LIN {X 0,Y 297.414,Z 212.275,A -85,B 0,C 180,E1 -16492.846,E2 -16492.846} C_VEL
LIN {X 0,Y 297.108,Z 216.721,A -85,B 0,C 180,E1 -16496.707,E2 -16496.707} C_VEL
LIN {X 0,Y 297.039,Z 218.831,A -85,B 0,C 180,E1 -16498.514,E2 -16498.514} C_VEL
LIN {X 0,Y 298.985,Z 230.293,A -85,B 0,C 180,E1 -16499.329,E2 -16499.329} C_VEL
LIN {X 0,Y 300.063,Z 238.045,A -85,B 0,C 180,E1 -16500.022,E2 -16500.022} C_VEL
LIN {X 0,Y 300.785,Z 244.745,A -85,B 0,C 180,E1 -16500.738,E2 -16500.738} C_VEL
LIN {X 0,Y 300.112,Z 253.295,A -85,B 0,C 180,E1 -16501.796,E2 -16501.796} C_VEL
LIN {X 0,Y 299.342,Z 261.65,A -85,B 0,C 180,E1 -16503.084,E2 -16503.084} C_VEL
LIN {X 0,Y 298.596,Z 269.147,A -85,B 0,C 180,E1 -16504.537,E2 -16504.537} C_VEL
LIN {X 0,Y 298.008,Z 275.588,A -85,B 0,C 180,E1 -16506.127,E2 -16506.127} C_VEL
LIN {X 0,Y 297.4,Z 281.322,A -85,B 0,C 180,E1 -16507.91,E2 -16507.91} C_VEL
LIN {X 0,Y 296.932,Z 285.817,A -85,B 0,C 180,E1 -16509.721,E2 -16509.721} C_VEL
LIN {X 0,Y 296.668,Z 289.117,A -85,B 0,C 180,E1 -16511.553,E2 -16511.553} C_VEL
LIN {X 0,Y 296.474,Z 291.311,A -85,B 0,C 180,E1 -16513.429,E2 -16513.429} C_VEL
LIN {X 0,Y 296.443,Z 292.469,A -85,B 0,C 180,E1 -16515.335,E2 -16515.335} C_VEL
LIN {X 0,Y 296.588,Z 292.583,A -85,B 0,C 180,E1 -16517.272,E2 -16517.272} C_VEL
LIN {X 0,Y 296.965,Z 291.615,A -85,B 0,C 180,E1 -16519.228,E2 -16519.228} C_VEL
LIN {X 0,Y 297.538,Z 289.488,A -85,B 0,C 180,E1 -16521.212,E2 -16521.212} C_VEL
LIN {X 0,Y 298.269,Z 285.912,A -85,B 0,C 180,E1 -16523.238,E2 -16523.238} C_VEL
LIN {X 0,Y 299.253,Z 280.84,A -85,B 0,C 180,E1 -16525.283,E2 -16525.283} C_VEL
LIN {X 0,Y 300.568,Z 273.927,A -85,B 0,C 180,E1 -16527.327,E2 -16527.327} C_VEL
LIN {X 0,Y 301.642,Z 267.542,A -85,B 0,C 180,E1 -16528.776,E2 -16528.776} C_VEL
LIN {X 0,Y 302.836,Z 260.472,A -85,B 0,C 180,E1 -16530.071,E2 -16530.071} C_VEL
LIN {X 0,Y 304.08,Z 251.263,A -85,B 0,C 180,E1 -16531.434,E2 -16531.434} C_VEL
LIN {X 0,Y 303.978,Z 248.011,A -85,B 0,C 180,E1 -16531.86,E2 -16531.86} C_VEL
LIN {X 0,Y 302.759,Z 239.813,A -85,B 0,C 180,E1 -16532.901,E2 -16532.901} C_VEL
LIN {X 0,Y 301.269,Z 232.79,A -85,B 0,C 180,E1 -16533.691,E2 -16533.691} C_VEL
LIN {X 0,Y 298.786,Z 224.127,A -85,B 0,C 180,E1 -16534.557,E2 -16534.557} C_VEL
LIN {X 0,Y 297.767,Z 220.447,A -85,B 0,C 180,E1 -16534.908,E2 -16534.908} C_VEL
LIN {X 0,Y 298.166,Z 216.073,A -85,B 0,C 180,E1 -16539.296,E2 -16539.296} C_VEL
LIN {X 0,Y 298.502,Z 213.292,A -85,B 0,C 180,E1 -16542.179,E2 -16542.179} C_VEL
LIN {X 0,Y 298.837,Z 210.683,A -85,B 0,C 180,E1 -16545.009,E2 -16545.009} C_VEL
LIN {X 0,Y 298.987,Z 208.224,A -85,B 0,C 180,E1 -16547.788,E2 -16547.788} C_VEL
LIN {X 0,Y 298.888,Z 204.918,A -85,B 0,C 180,E1 -16551.891,E2 -16551.891} C_VEL
LIN {X 0,Y 298.802,Z 204.086,A -85,B 0,C 180,E1 -16553.247,E2 -16553.247} C_VEL
LIN {X 0,Y 298.84,Z 204.074,A -85,B 0,C 180,E1 -16557.531,E2 -16557.531} C_VEL
LIN {X 0,Y 298.211,Z 204.153,A -85,B 0,C 180,E1 -16558.658,E2 -16558.658} C_VEL
LIN {X 0,Y 295.396,Z 204.503,A -85,B 0,C 180,E1 -16560.493,E2 -16560.493} C_VEL
LIN {X 0,Y 292.054,Z 204.917,A -85,B 0,C 180,E1 -16562.745,E2 -16562.745} C_VEL
LIN {X 0,Y 291.638,Z 204.968,A -85,B 0,C 180,E1 -16563.524,E2 -16563.524} C_VEL
LIN {X 0,Y 291.725,Z 204.961,A -85,B 0,C 180,E1 -16566.92,E2 -16566.92} C_VEL
LIN {X 0,Y 291.569,Z 204.98,A -85,B 0,C 180,E1 -16569.715,E2 -16569.715} C_VEL
LIN {X 0,Y 291.524,Z 204.986,A -85,B 0,C 180,E1 -16573.951,E2 -16573.951} C_VEL
LIN {X 0,Y 291.489,Z 204.99,A -85,B 0,C 180,E1 -16576.819,E2 -16576.819} C_VEL
LIN {X 0,Y 291.453,Z 204.994,A -85,B 0,C 180,E1 -16579.876,E2 -16579.876} C_VEL
LIN {X 0,Y 291.403,Z 205.001,A -85,B 0,C 180,E1 -16584.206,E2 -16584.206} C_VEL
LIN {X 0,Y 291.425,Z 204.997,A -85,B 0,C 180,E1 -16587.272,E2 -16587.272} C_VEL
LIN {X 0,Y 291.34,Z 205.007,A -85,B 0,C 180,E1 -16590.438,E2 -16590.438} C_VEL
LIN {X 0,Y 291.347,Z 205.006,A -85,B 0,C 180,E1 -16593.699,E2 -16593.699} C_VEL
LIN {X 0,Y 291.383,Z 205.003,A -85,B 0,C 180,E1 -16597.256,E2 -16597.256} C_VEL
LIN {X 0,Y 291.336,Z 205.011,A -85,B 0,C 180,E1 -16600.643,E2 -16600.643} C_VEL
LIN {X 0,Y 291.356,Z 205.078,A -85,B 0,C 180,E1 -16602.79,E2 -16602.79} C_VEL
LIN {X 0,Y 291.895,Z 208.233,A -85,B 0,C 180,E1 -16606.247,E2 -16606.247} C_VEL
LIN {X 0,Y 292.713,Z 212.344,A -85,B 0,C 180,E1 -16610.204,E2 -16610.204} C_VEL
LIN {X 0,Y 293.351,Z 215.803,A -85,B 0,C 180,E1 -16613.206,E2 -16613.206} C_VEL
LIN {X 0,Y 294.12,Z 220.258,A -85,B 0,C 180,E1 -16616.755,E2 -16616.755} C_VEL
LIN {X 0,Y 294.047,Z 222.378,A -85,B 0,C 180,E1 -16618.277,E2 -16618.277} C_VEL
LIN {X 0,Y 293.07,Z 226.935,A -85,B 0,C 180,E1 -16621.34,E2 -16621.34} C_VEL
LIN {X 0,Y 291.758,Z 233.962,A -85,B 0,C 180,E1 -16625.827,E2 -16625.827} C_VEL
LIN {X 0,Y 291.109,Z 238.512,A -85,B 0,C 180,E1 -16628.63,E2 -16628.63} C_VEL
LIN {X 0,Y 293.61,Z 250.168,A -85,B 0,C 180,E1 -16629.573,E2 -16629.573} C_VEL
LIN {X 0,Y 295.041,Z 259.692,A -85,B 0,C 180,E1 -16630.52,E2 -16630.52} C_VEL
LIN {X 0,Y 295.682,Z 269.392,A -85,B 0,C 180,E1 -16631.644,E2 -16631.644} C_VEL
LIN {X 0,Y 295.708,Z 276.379,A -85,B 0,C 180,E1 -16632.581,E2 -16632.581} C_VEL
LIN {X 0,Y 295.117,Z 282.939,A -85,B 0,C 180,E1 -16633.573,E2 -16633.573} C_VEL
LIN {X 0,Y 293.912,Z 289.657,A -85,B 0,C 180,E1 -16634.75,E2 -16634.75} C_VEL
LIN {X 0,Y 292.758,Z 296.048,A -85,B 0,C 180,E1 -16636.11,E2 -16636.11} C_VEL
LIN {X 0,Y 291.865,Z 301.377,A -85,B 0,C 180,E1 -16637.484,E2 -16637.484} C_VEL
LIN {X 0,Y 291.099,Z 305.839,A -85,B 0,C 180,E1 -16638.864,E2 -16638.864} C_VEL
LIN {X 0,Y 290.259,Z 311.111,A -85,B 0,C 180,E1 -16640.945,E2 -16640.945} C_VEL
LIN {X 0,Y 289.716,Z 315.016,A -85,B 0,C 180,E1 -16643.034,E2 -16643.034} C_VEL
LIN {X 0,Y 289.519,Z 316.836,A -85,B 0,C 180,E1 -16644.428,E2 -16644.428} C_VEL
LIN {X 0,Y 289.499,Z 318.156,A -85,B 0,C 180,E1 -16645.824,E2 -16645.824} C_VEL
LIN {X 0,Y 289.515,Z 318.987,A -85,B 0,C 180,E1 -16647.217,E2 -16647.217} C_VEL
LIN {X 0,Y 289.513,Z 319.327,A -85,B 0,C 180,E1 -16648.609,E2 -16648.609} C_VEL
LIN {X 0,Y 289.584,Z 319.077,A -85,B 0,C 180,E1 -16650,E2 -16650} C_VEL
LIN {X 0,Y 289.546,Z 318.288,A -85,B 0,C 180,E1 -16651.391,E2 -16651.391} C_VEL
LIN {X 0,Y 289.545,Z 316.998,A -85,B 0,C 180,E1 -16652.783,E2 -16652.783} C_VEL
LIN {X 0,Y 289.601,Z 315.181,A -85,B 0,C 180,E1 -16654.175,E2 -16654.175} C_VEL
LIN {X 0,Y 289.611,Z 311.418,A -85,B 0,C 180,E1 -16656.2,E2 -16656.2} C_VEL
LIN {X 0,Y 289.838,Z 307.852,A -85,B 0,C 180,E1 -16657.664,E2 -16657.664} C_VEL
LIN {X 0,Y 290.258,Z 302.518,A -85,B 0,C 180,E1 -16659.407,E2 -16659.407} C_VEL
LIN {X 0,Y 290.833,Z 295.827,A -85,B 0,C 180,E1 -16661.147,E2 -16661.147} C_VEL
LIN {X 0,Y 291.684,Z 287.227,A -85,B 0,C 180,E1 -16662.878,E2 -16662.878} C_VEL
LIN {X 0,Y 292.473,Z 279.712,A -85,B 0,C 180,E1 -16664.082,E2 -16664.082} C_VEL
LIN {X 0,Y 292.816,Z 273.278,A -85,B 0,C 180,E1 -16664.953,E2 -16664.953} C_VEL
LIN {X 0,Y 292.351,Z 264.646,A -85,B 0,C 180,E1 -16665.931,E2 -16665.931} C_VEL
LIN {X 0,Y 291.763,Z 256.683,A -85,B 0,C 180,E1 -16666.667,E2 -16666.667} C_VEL
LIN {X 0,Y 290.887,Z 246.792,A -85,B 0,C 180,E1 -16667.374,E2 -16667.374} C_VEL
LIN {X 0,Y 290.186,Z 239.923,A -85,B 0,C 180,E1 -16667.804,E2 -16667.804} C_VEL
LIN {X 0,Y 290.881,Z 232.782,A -85,B 0,C 180,E1 -16671.994,E2 -16671.994} C_VEL
LIN {X 0,Y 291.85,Z 225.39,A -85,B 0,C 180,E1 -16676.385,E2 -16676.385} C_VEL
LIN {X 0,Y 292.868,Z 218.975,A -85,B 0,C 180,E1 -16680.261,E2 -16680.261} C_VEL
LIN {X 0,Y 293.266,Z 216.446,A -85,B 0,C 180,E1 -16681.818,E2 -16681.818} C_VEL
LIN {X 0,Y 292.826,Z 212.59,A -85,B 0,C 180,E1 -16684.334,E2 -16684.334} C_VEL
LIN {X 0,Y 292.012,Z 208.048,A -85,B 0,C 180,E1 -16687.416,E2 -16687.416} C_VEL
LIN {X 0,Y 291.415,Z 205.002,A -85,B 0,C 180,E1 -16689.691,E2 -16689.691} C_VEL
LIN {X 0,Y 291.313,Z 205.008,A -85,B 0,C 180,E1 -16693.633,E2 -16693.633} C_VEL
LIN {X 0,Y 291.304,Z 205.008,A -85,B 0,C 180,E1 -16697.504,E2 -16697.504} C_VEL
LIN {X 0,Y 291.343,Z 205.004,A -85,B 0,C 180,E1 -16701.156,E2 -16701.156} C_VEL
LIN {X 0,Y 291.359,Z 205.002,A -85,B 0,C 180,E1 -16704.625,E2 -16704.625} C_VEL
LIN {X 0,Y 291.375,Z 205.004,A -85,B 0,C 180,E1 -16707.95,E2 -16707.95} C_VEL
LIN {X 0,Y 291.382,Z 204.999,A -85,B 0,C 180,E1 -16711.157,E2 -16711.157} C_VEL
LIN {X 0,Y 291.42,Z 204.996,A -85,B 0,C 180,E1 -16714.271,E2 -16714.271} C_VEL
LIN {X 0,Y 291.379,Z 205.001,A -85,B 0,C 180,E1 -16717.298,E2 -16717.298} C_VEL
LIN {X 0,Y 291.462,Z 204.989,A -85,B 0,C 180,E1 -16720.269,E2 -16720.269} C_VEL
LIN {X 0,Y 291.56,Z 204.977,A -85,B 0,C 180,E1 -16724.623,E2 -16724.623} C_VEL
LIN {X 0,Y 291.533,Z 204.98,A -85,B 0,C 180,E1 -16728.879,E2 -16728.879} C_VEL
LIN {X 0,Y 291.671,Z 204.966,A -85,B 0,C 180,E1 -16731.686,E2 -16731.686} C_VEL
LIN {X 0,Y 291.626,Z 204.969,A -85,B 0,C 180,E1 -16734.467,E2 -16734.467} C_VEL
LIN {X 0,Y 291.892,Z 204.935,A -85,B 0,C 180,E1 -16738.619,E2 -16738.619} C_VEL
LIN {X 0,Y 291.89,Z 204.939,A -85,B 0,C 180,E1 -16741.378,E2 -16741.378} C_VEL
LIN {X 0,Y 291.725,Z 204.96,A -85,B 0,C 180,E1 -16746.917,E2 -16746.917} C_VEL
LIN {X 0,Y 291.57,Z 204.976,A -85,B 0,C 180,E1 -16749.713,E2 -16749.713} C_VEL
LIN {X 0,Y 291.517,Z 204.982,A -85,B 0,C 180,E1 -16753.949,E2 -16753.949} C_VEL
LIN {X 0,Y 291.429,Z 204.997,A -85,B 0,C 180,E1 -16756.82,E2 -16756.82} C_VEL
LIN {X 0,Y 291.424,Z 204.994,A -85,B 0,C 180,E1 -16759.859,E2 -16759.859} C_VEL
LIN {X 0,Y 291.383,Z 205,A -85,B 0,C 180,E1 -16764.205,E2 -16764.205} C_VEL
LIN {X 0,Y 291.422,Z 204.994,A -85,B 0,C 180,E1 -16767.27,E2 -16767.27} C_VEL
LIN {X 0,Y 291.336,Z 205.008,A -85,B 0,C 180,E1 -16770.435,E2 -16770.435} C_VEL
LIN {X 0,Y 291.343,Z 205.004,A -85,B 0,C 180,E1 -16773.697,E2 -16773.697} C_VEL
LIN {X 0,Y 291.391,Z 204.998,A -85,B 0,C 180,E1 -16777.257,E2 -16777.257} C_VEL
LIN {X 0,Y 291.33,Z 205.006,A -85,B 0,C 180,E1 -16780.641,E2 -16780.641} C_VEL
LIN {X 0,Y 291.286,Z 205.013,A -85,B 0,C 180,E1 -16784.4,E2 -16784.4} C_VEL
LIN {X 0,Y 291.321,Z 205.007,A -85,B 0,C 180,E1 -16788.403,E2 -16788.403} C_VEL
LIN {X 0,Y 291.358,Z 205.002,A -85,B 0,C 180,E1 -16791.159,E2 -16791.159} C_VEL
LIN {X 0,Y 291.356,Z 205.002,A -85,B 0,C 180,E1 -16794.625,E2 -16794.625} C_VEL
LIN {X 0,Y 291.367,Z 205.003,A -85,B 0,C 180,E1 -16797.95,E2 -16797.95} C_VEL
LIN {X 0,Y 291.384,Z 205.001,A -85,B 0,C 180,E1 -16801.158,E2 -16801.158} C_VEL
LIN {X 0,Y 291.414,Z 204.994,A -85,B 0,C 180,E1 -16804.271,E2 -16804.271} C_VEL
LIN {X 0,Y 291.374,Z 205.004,A -85,B 0,C 180,E1 -16807.299,E2 -16807.299} C_VEL
LIN {X 0,Y 291.451,Z 204.99,A -85,B 0,C 180,E1 -16810.269,E2 -16810.269} C_VEL
LIN {X 0,Y 291.548,Z 204.979,A -85,B 0,C 180,E1 -16814.623,E2 -16814.623} C_VEL
LIN {X 0,Y 291.531,Z 204.984,A -85,B 0,C 180,E1 -16818.88,E2 -16818.88} C_VEL
LIN {X 0,Y 291.701,Z 204.959,A -85,B 0,C 180,E1 -16821.688,E2 -16821.688} C_VEL
LIN {X 0,Y 291.623,Z 204.97,A -85,B 0,C 180,E1 -16824.468,E2 -16824.468} C_VEL
LIN {X 0,Y 291.883,Z 204.94,A -85,B 0,C 180,E1 -16828.62,E2 -16828.62} C_VEL
LIN {X 0,Y 291.882,Z 204.937,A -85,B 0,C 180,E1 -16831.379,E2 -16831.379} C_VEL
LIN {X 0,Y 291.744,Z 204.955,A -85,B 0,C 180,E1 -16836.918,E2 -16836.918} C_VEL
LIN {X 0,Y 291.618,Z 204.969,A -85,B 0,C 180,E1 -16839.712,E2 -16839.712} C_VEL
LIN {X 0,Y 291.27,Z 205.015,A -85,B 0,C 180,E1 -16843.962,E2 -16843.962} C_VEL
LIN {X 0,Y 290.981,Z 205.27,A -85,B 0,C 180,E1 -16845.766,E2 -16845.766} C_VEL
LIN {X 0,Y 290.55,Z 209.635,A -85,B 0,C 180,E1 -16849.794,E2 -16849.794} C_VEL
LIN {X 0,Y 290.327,Z 213.294,A -85,B 0,C 180,E1 -16853.097,E2 -16853.097} C_VEL
LIN {X 0,Y 290.083,Z 216.893,A -85,B 0,C 180,E1 -16856.313,E2 -16856.313} C_VEL
LIN {X 0,Y 289.97,Z 219.046,A -85,B 0,C 180,E1 -16858.204,E2 -16858.204} C_VEL
LIN {X 0,Y 291.957,Z 230.689,A -85,B 0,C 180,E1 -16859.057,E2 -16859.057} C_VEL
LIN {X 0,Y 293.29,Z 240.396,A -85,B 0,C 180,E1 -16859.972,E2 -16859.972} C_VEL
LIN {X 0,Y 293.767,Z 245.455,A -85,B 0,C 180,E1 -16860.546,E2 -16860.546} C_VEL
LIN {X 0,Y 293.108,Z 253.829,A -85,B 0,C 180,E1 -16861.615,E2 -16861.615} C_VEL
LIN {X 0,Y 292.351,Z 261.767,A -85,B 0,C 180,E1 -16862.869,E2 -16862.869} C_VEL
LIN {X 0,Y 291.509,Z 269.966,A -85,B 0,C 180,E1 -16864.511,E2 -16864.511} C_VEL
LIN {X 0,Y 290.871,Z 276.61,A -85,B 0,C 180,E1 -16866.222,E2 -16866.222} C_VEL
LIN {X 0,Y 290.387,Z 281.151,A -85,B 0,C 180,E1 -16867.669,E2 -16867.669} C_VEL
LIN {X 0,Y 289.983,Z 284.899,A -85,B 0,C 180,E1 -16869.148,E2 -16869.148} C_VEL
LIN {X 0,Y 289.64,Z 288.377,A -85,B 0,C 180,E1 -16870.93,E2 -16870.93} C_VEL
LIN {X 0,Y 289.389,Z 291.434,A -85,B 0,C 180,E1 -16873.236,E2 -16873.236} C_VEL
LIN {X 0,Y 289.347,Z 292.738,A -85,B 0,C 180,E1 -16875.222,E2 -16875.222} C_VEL
LIN {X 0,Y 289.485,Z 292.971,A -85,B 0,C 180,E1 -16877.176,E2 -16877.176} C_VEL
LIN {X 0,Y 289.852,Z 292.183,A -85,B 0,C 180,E1 -16879.108,E2 -16879.108} C_VEL
LIN {X 0,Y 290.404,Z 290.396,A -85,B 0,C 180,E1 -16881.009,E2 -16881.009} C_VEL
LIN {X 0,Y 290.99,Z 287.65,A -85,B 0,C 180,E1 -16882.859,E2 -16882.859} C_VEL
LIN {X 0,Y 291.979,Z 283.171,A -85,B 0,C 180,E1 -16884.923,E2 -16884.923} C_VEL
LIN {X 0,Y 292.915,Z 278.606,A -85,B 0,C 180,E1 -16886.508,E2 -16886.508} C_VEL
LIN {X 0,Y 293.915,Z 273.358,A -85,B 0,C 180,E1 -16887.972,E2 -16887.972} C_VEL
LIN {X 0,Y 294.951,Z 267.831,A -85,B 0,C 180,E1 -16889.236,E2 -16889.236} C_VEL
LIN {X 0,Y 296.026,Z 261.783,A -85,B 0,C 180,E1 -16890.384,E2 -16890.384} C_VEL
LIN {X 0,Y 297.139,Z 254.197,A -85,B 0,C 180,E1 -16891.578,E2 -16891.578} C_VEL
LIN {X 0,Y 297.373,Z 250.008,A -85,B 0,C 180,E1 -16892.177,E2 -16892.177} C_VEL
LIN {X 0,Y 296.132,Z 240.963,A -85,B 0,C 180,E1 -16893.389,E2 -16893.389} C_VEL
LIN {X 0,Y 294.297,Z 232.789,A -85,B 0,C 180,E1 -16894.354,E2 -16894.354} C_VEL
LIN {X 0,Y 291.629,Z 223.663,A -85,B 0,C 180,E1 -16895.295,E2 -16895.295} C_VEL
LIN {X 0,Y 290.755,Z 220.769,A -85,B 0,C 180,E1 -16895.597,E2 -16895.597} C_VEL
LIN {X 0,Y 291.069,Z 217.689,A -85,B 0,C 180,E1 -16898.767,E2 -16898.767} C_VEL
LIN {X 0,Y 291.442,Z 214.883,A -85,B 0,C 180,E1 -16901.732,E2 -16901.732} C_VEL
LIN {X 0,Y 291.801,Z 212.252,A -85,B 0,C 180,E1 -16904.638,E2 -16904.638} C_VEL
LIN {X 0,Y 292.004,Z 209.785,A -85,B 0,C 180,E1 -16907.491,E2 -16907.491} C_VEL
LIN {X 0,Y 291.933,Z 206.457,A -85,B 0,C 180,E1 -16911.696,E2 -16911.696} C_VEL
LIN {X 0,Y 291.819,Z 205.463,A -85,B 0,C 180,E1 -16913.085,E2 -16913.085} C_VEL
LIN {X 0,Y 291.632,Z 204.979,A -85,B 0,C 180,E1 -16914.47,E2 -16914.47} C_VEL
LIN {X 0,Y 291.891,Z 204.941,A -85,B 0,C 180,E1 -16918.622,E2 -16918.622} C_VEL
LIN {X 0,Y 291.891,Z 204.937,A -85,B 0,C 180,E1 -16921.381,E2 -16921.381} C_VEL
LIN {X 0,Y 291.638,Z 204.968,A -85,B 0,C 180,E1 -16923.524,E2 -16923.524} C_VEL
LIN {X 0,Y 290.865,Z 205.068,A -85,B 0,C 180,E1 -16924.677,E2 -16924.677} C_VEL
LIN {X 0,Y 288.043,Z 205.419,A -85,B 0,C 180,E1 -16926.557,E2 -16926.557} C_VEL
LIN {X 0,Y 285.693,Z 205.712,A -85,B 0,C 180,E1 -16928.083,E2 -16928.083} C_VEL
LIN {X 0,Y 284.648,Z 205.841,A -85,B 0,C 180,E1 -16929.262,E2 -16929.262} C_VEL
LIN {X 0,Y 284.539,Z 205.854,A -85,B 0,C 180,E1 -16929.662,E2 -16929.662} C_VEL
LIN {X 0,Y 284.484,Z 205.861,A -85,B 0,C 180,E1 -16934.304,E2 -16934.304} C_VEL
LIN {X 0,Y 284.428,Z 205.869,A -85,B 0,C 180,E1 -16937.249,E2 -16937.249} C_VEL
LIN {X 0,Y 284.381,Z 205.874,A -85,B 0,C 180,E1 -16940.243,E2 -16940.243} C_VEL
LIN {X 0,Y 284.372,Z 205.876,A -85,B 0,C 180,E1 -16943.876,E2 -16943.876} C_VEL
LIN {X 0,Y 284.4,Z 205.873,A -85,B 0,C 180,E1 -16947.175,E2 -16947.175} C_VEL
LIN {X 0,Y 284.298,Z 205.884,A -85,B 0,C 180,E1 -16951.275,E2 -16951.275} C_VEL
LIN {X 0,Y 284.343,Z 205.878,A -85,B 0,C 180,E1 -16955.349,E2 -16955.349} C_VEL
LIN {X 0,Y 284.321,Z 205.884,A -85,B 0,C 180,E1 -16958.169,E2 -16958.169} C_VEL
LIN {X 0,Y 284.314,Z 206.084,A -85,B 0,C 180,E1 -16961.869,E2 -16961.869} C_VEL
LIN {X 0,Y 284.717,Z 208.103,A -85,B 0,C 180,E1 -16964.288,E2 -16964.288} C_VEL
LIN {X 0,Y 285.381,Z 211.939,A -85,B 0,C 180,E1 -16968.324,E2 -16968.324} C_VEL
LIN {X 0,Y 286.208,Z 216.023,A -85,B 0,C 180,E1 -16972.129,E2 -16972.129} C_VEL
LIN {X 0,Y 287.064,Z 221.078,A -85,B 0,C 180,E1 -16976.347,E2 -16976.347} C_VEL
LIN {X 0,Y 287.213,Z 222.474,A -85,B 0,C 180,E1 -16977.43,E2 -16977.43} C_VEL
LIN {X 0,Y 286.26,Z 227.01,A -85,B 0,C 180,E1 -16980.592,E2 -16980.592} C_VEL
LIN {X 0,Y 285.085,Z 232.803,A -85,B 0,C 180,E1 -16984.443,E2 -16984.443} C_VEL
LIN {X 0,Y 284.198,Z 238.221,A -85,B 0,C 180,E1 -16987.916,E2 -16987.916} C_VEL
LIN {X 0,Y 286.946,Z 250.877,A -85,B 0,C 180,E1 -16989.001,E2 -16989.001} C_VEL
LIN {X 0,Y 288.401,Z 260.855,A -85,B 0,C 180,E1 -16990.052,E2 -16990.052} C_VEL
LIN {X 0,Y 288.953,Z 268.817,A -85,B 0,C 180,E1 -16991.017,E2 -16991.017} C_VEL
LIN {X 0,Y 288.943,Z 277.148,A -85,B 0,C 180,E1 -16992.186,E2 -16992.186} C_VEL
LIN {X 0,Y 288.335,Z 283.349,A -85,B 0,C 180,E1 -16993.175,E2 -16993.175} C_VEL
LIN {X 0,Y 286.741,Z 291.629,A -85,B 0,C 180,E1 -16994.723,E2 -16994.723} C_VEL
LIN {X 0,Y 285.43,Z 299.052,A -85,B 0,C 180,E1 -16996.473,E2 -16996.473} C_VEL
LIN {X 0,Y 284.316,Z 304.884,A -85,B 0,C 180,E1 -16998.233,E2 -16998.233} C_VEL
LIN {X 0,Y 283.501,Z 309.507,A -85,B 0,C 180,E1 -17000.007,E2 -17000.007} C_VEL
LIN {X 0,Y 282.789,Z 313.708,A -85,B 0,C 180,E1 -17002.144,E2 -17002.144} C_VEL
LIN {X 0,Y 282.445,Z 316.653,A -85,B 0,C 180,E1 -17004.288,E2 -17004.288} C_VEL
LIN {X 0,Y 282.402,Z 317.909,A -85,B 0,C 180,E1 -17005.719,E2 -17005.719} C_VEL
LIN {X 0,Y 282.441,Z 318.684,A -85,B 0,C 180,E1 -17007.148,E2 -17007.148} C_VEL
LIN {X 0,Y 282.431,Z 318.978,A -85,B 0,C 180,E1 -17008.574,E2 -17008.574} C_VEL
LIN {X 0,Y 282.497,Z 318.717,A -85,B 0,C 180,E1 -17010,E2 -17010} C_VEL
LIN {X 0,Y 282.463,Z 317.878,A -85,B 0,C 180,E1 -17011.426,E2 -17011.426} C_VEL
LIN {X 0,Y 282.474,Z 316.533,A -85,B 0,C 180,E1 -17012.853,E2 -17012.853} C_VEL
LIN {X 0,Y 282.458,Z 313.396,A -85,B 0,C 180,E1 -17015.063,E2 -17015.063} C_VEL
LIN {X 0,Y 282.673,Z 309.101,A -85,B 0,C 180,E1 -17017.141,E2 -17017.141} C_VEL
LIN {X 0,Y 283.028,Z 304.133,A -85,B 0,C 180,E1 -17018.928,E2 -17018.928} C_VEL
LIN {X 0,Y 283.552,Z 297.841,A -85,B 0,C 180,E1 -17020.713,E2 -17020.713} C_VEL
LIN {X 0,Y 284.134,Z 291.663,A -85,B 0,C 180,E1 -17022.137,E2 -17022.137} C_VEL
LIN {X 0,Y 284.737,Z 285.152,A -85,B 0,C 180,E1 -17023.38,E2 -17023.38} C_VEL
LIN {X 0,Y 285.483,Z 278.51,A -85,B 0,C 180,E1 -17024.434,E2 -17024.434} C_VEL
LIN {X 0,Y 285.756,Z 273.371,A -85,B 0,C 180,E1 -17025.148,E2 -17025.148} C_VEL
LIN {X 0,Y 285.299,Z 264.256,A -85,B 0,C 180,E1 -17026.209,E2 -17026.209} C_VEL
LIN {X 0,Y 284.589,Z 254.94,A -85,B 0,C 180,E1 -17027.073,E2 -17027.073} C_VEL
LIN {X 0,Y 283.716,Z 245.299,A -85,B 0,C 180,E1 -17027.758,E2 -17027.758} C_VEL
LIN {X 0,Y 283.146,Z 239.755,A -85,B 0,C 180,E1 -17028.075,E2 -17028.075} C_VEL
LIN {X 0,Y 283.912,Z 232.315,A -85,B 0,C 180,E1 -17032.563,E2 -17032.563} C_VEL
LIN {X 0,Y 284.778,Z 226.072,A -85,B 0,C 180,E1 -17036.374,E2 -17036.374} C_VEL
LIN {X 0,Y 285.916,Z 219.211,A -85,B 0,C 180,E1 -17040.646,E2 -17040.646} C_VEL
LIN {X 0,Y 286.229,Z 217.286,A -85,B 0,C 180,E1 -17041.864,E2 -17041.864} C_VEL
LIN {X 0,Y 285.775,Z 213.4,A -85,B 0,C 180,E1 -17044.447,E2 -17044.447} C_VEL
LIN {X 0,Y 284.794,Z 208.19,A -85,B 0,C 180,E1 -17048.093,E2 -17048.093} C_VEL
LIN {X 0,Y 284.363,Z 205.881,A -85,B 0,C 180,E1 -17049.868,E2 -17049.868} C_VEL
LIN {X 0,Y 284.25,Z 205.89,A -85,B 0,C 180,E1 -17054.19,E2 -17054.19} C_VEL
LIN {X 0,Y 284.266,Z 205.888,A -85,B 0,C 180,E1 -17058.122,E2 -17058.122} C_VEL
LIN {X 0,Y 284.304,Z 205.883,A -85,B 0,C 180,E1 -17061.829,E2 -17061.829} C_VEL
LIN {X 0,Y 284.311,Z 205.879,A -85,B 0,C 180,E1 -17065.35,E2 -17065.35} C_VEL
LIN {X 0,Y 284.298,Z 205.882,A -85,B 0,C 180,E1 -17068.725,E2 -17068.725} C_VEL
LIN {X 0,Y 284.401,Z 205.868,A -85,B 0,C 180,E1 -17072.826,E2 -17072.826} C_VEL
LIN {X 0,Y 284.338,Z 205.877,A -85,B 0,C 180,E1 -17076.703,E2 -17076.703} C_VEL
LIN {X 0,Y 284.404,Z 205.869,A -85,B 0,C 180,E1 -17081.261,E2 -17081.261} C_VEL
LIN {X 0,Y 284.497,Z 205.857,A -85,B 0,C 180,E1 -17084.458,E2 -17084.458} C_VEL
LIN {X 0,Y 284.487,Z 205.857,A -85,B 0,C 180,E1 -17088.6,E2 -17088.6} C_VEL
LIN {X 0,Y 284.626,Z 205.845,A -85,B 0,C 180,E1 -17091.479,E2 -17091.479} C_VEL
LIN {X 0,Y 284.596,Z 205.844,A -85,B 0,C 180,E1 -17094.33,E2 -17094.33} C_VEL
LIN {X 0,Y 284.858,Z 205.811,A -85,B 0,C 180,E1 -17098.585,E2 -17098.585} C_VEL
LIN {X 0,Y 284.856,Z 205.815,A -85,B 0,C 180,E1 -17101.413,E2 -17101.413} C_VEL
LIN {X 0,Y 284.676,Z 205.838,A -85,B 0,C 180,E1 -17107.089,E2 -17107.089} C_VEL
LIN {X 0,Y 284.516,Z 205.854,A -85,B 0,C 180,E1 -17109.956,E2 -17109.956} C_VEL
LIN {X 0,Y 284.465,Z 205.861,A -85,B 0,C 180,E1 -17114.302,E2 -17114.302} C_VEL
LIN {X 0,Y 284.341,Z 205.881,A -85,B 0,C 180,E1 -17118.741,E2 -17118.741} C_VEL
LIN {X 0,Y 284.312,Z 205.879,A -85,B 0,C 180,E1 -17121.763,E2 -17121.763} C_VEL
LIN {X 0,Y 284.338,Z 205.878,A -85,B 0,C 180,E1 -17124.845,E2 -17124.845} C_VEL
LIN {X 0,Y 284.331,Z 205.879,A -85,B 0,C 180,E1 -17128.009,E2 -17128.009} C_VEL
LIN {X 0,Y 284.295,Z 205.881,A -85,B 0,C 180,E1 -17131.273,E2 -17131.273} C_VEL
LIN {X 0,Y 284.359,Z 205.874,A -85,B 0,C 180,E1 -17135.352,E2 -17135.352} C_VEL
LIN {X 0,Y 284.32,Z 205.883,A -85,B 0,C 180,E1 -17138.166,E2 -17138.166} C_VEL
LIN {X 0,Y 284.266,Z 205.89,A -85,B 0,C 180,E1 -17142.123,E2 -17142.123} C_VEL
LIN {X 0,Y 284.251,Z 205.89,A -85,B 0,C 180,E1 -17146.188,E2 -17146.188} C_VEL
LIN {X 0,Y 284.302,Z 205.884,A -85,B 0,C 180,E1 -17150.022,E2 -17150.022} C_VEL
LIN {X 0,Y 284.329,Z 205.882,A -85,B 0,C 180,E1 -17153.613,E2 -17153.613} C_VEL
LIN {X 0,Y 284.302,Z 205.881,A -85,B 0,C 180,E1 -17157.188,E2 -17157.188} C_VEL
LIN {X 0,Y 284.356,Z 205.874,A -85,B 0,C 180,E1 -17160.375,E2 -17160.375} C_VEL
LIN {X 0,Y 284.375,Z 205.875,A -85,B 0,C 180,E1 -17163.586,E2 -17163.586} C_VEL
LIN {X 0,Y 284.359,Z 205.874,A -85,B 0,C 180,E1 -17166.706,E2 -17166.706} C_VEL
LIN {X 0,Y 284.397,Z 205.874,A -85,B 0,C 180,E1 -17171.261,E2 -17171.261} C_VEL
LIN {X 0,Y 284.485,Z 205.858,A -85,B 0,C 180,E1 -17174.458,E2 -17174.458} C_VEL
LIN {X 0,Y 284.483,Z 205.86,A -85,B 0,C 180,E1 -17178.601,E2 -17178.601} C_VEL
LIN {X 0,Y 284.651,Z 205.837,A -85,B 0,C 180,E1 -17181.481,E2 -17181.481} C_VEL
LIN {X 0,Y 284.593,Z 205.845,A -85,B 0,C 180,E1 -17184.331,E2 -17184.331} C_VEL
LIN {X 0,Y 284.848,Z 205.816,A -85,B 0,C 180,E1 -17188.586,E2 -17188.586} C_VEL
LIN {X 0,Y 284.848,Z 205.813,A -85,B 0,C 180,E1 -17191.414,E2 -17191.414} C_VEL
LIN {X 0,Y 284.697,Z 205.832,A -85,B 0,C 180,E1 -17197.09,E2 -17197.09} C_VEL
LIN {X 0,Y 284.536,Z 205.852,A -85,B 0,C 180,E1 -17199.956,E2 -17199.956} C_VEL
LIN {X 0,Y 284.184,Z 205.9,A -85,B 0,C 180,E1 -17204.318,E2 -17204.318} C_VEL
LIN {X 0,Y 283.913,Z 206.159,A -85,B 0,C 180,E1 -17205.801,E2 -17205.801} C_VEL
LIN {X 0,Y 283.423,Z 210.951,A -85,B 0,C 180,E1 -17210.313,E2 -17210.313} C_VEL
LIN {X 0,Y 283.234,Z 214.299,A -85,B 0,C 180,E1 -17213.391,E2 -17213.391} C_VEL
LIN {X 0,Y 282.902,Z 219.348,A -85,B 0,C 180,E1 -17217.915,E2 -17217.915} C_VEL
LIN {X 0,Y 284.843,Z 230.795,A -85,B 0,C 180,E1 -17218.759,E2 -17218.759} C_VEL
LIN {X 0,Y 286.122,Z 239.804,A -85,B 0,C 180,E1 -17219.619,E2 -17219.619} C_VEL
LIN {X 0,Y 286.765,Z 245.982,A -85,B 0,C 180,E1 -17220.33,E2 -17220.33} C_VEL
LIN {X 0,Y 286.062,Z 254.633,A -85,B 0,C 180,E1 -17221.471,E2 -17221.471} C_VEL
LIN {X 0,Y 285.085,Z 264.092,A -85,B 0,C 180,E1 -17223.055,E2 -17223.055} C_VEL
LIN {X 0,Y 284.322,Z 271.408,A -85,B 0,C 180,E1 -17224.647,E2 -17224.647} C_VEL
LIN {X 0,Y 283.702,Z 278.118,A -85,B 0,C 180,E1 -17226.48,E2 -17226.48} C_VEL
LIN {X 0,Y 283.086,Z 283.518,A -85,B 0,C 180,E1 -17228.364,E2 -17228.364} C_VEL
LIN {X 0,Y 282.636,Z 287.569,A -85,B 0,C 180,E1 -17230.279,E2 -17230.279} C_VEL
LIN {X 0,Y 282.391,Z 290.5,A -85,B 0,C 180,E1 -17232.218,E2 -17232.218} C_VEL
LIN {X 0,Y 282.26,Z 292.417,A -85,B 0,C 180,E1 -17234.2,E2 -17234.2} C_VEL
LIN {X 0,Y 282.302,Z 293.311,A -85,B 0,C 180,E1 -17236.217,E2 -17236.217} C_VEL
LIN {X 0,Y 282.586,Z 293.145,A -85,B 0,C 180,E1 -17238.254,E2 -17238.254} C_VEL
LIN {X 0,Y 283.083,Z 291.801,A -85,B 0,C 180,E1 -17240.32,E2 -17240.32} C_VEL
LIN {X 0,Y 283.751,Z 289.185,A -85,B 0,C 180,E1 -17242.427,E2 -17242.427} C_VEL
LIN {X 0,Y 284.268,Z 287.222,A -85,B 0,C 180,E1 -17243.606,E2 -17243.606} C_VEL
LIN {X 0,Y 285.188,Z 283.051,A -85,B 0,C 180,E1 -17245.475,E2 -17245.475} C_VEL
LIN {X 0,Y 286.38,Z 277.645,A -85,B 0,C 180,E1 -17247.325,E2 -17247.325} C_VEL
LIN {X 0,Y 287.782,Z 270.83,A -85,B 0,C 180,E1 -17249.148,E2 -17249.148} C_VEL
LIN {X 0,Y 289.259,Z 262.987,A -85,B 0,C 180,E1 -17250.749,E2 -17250.749} C_VEL
LIN {X 0,Y 290.523,Z 254.995,A -85,B 0,C 180,E1 -17252.052,E2 -17252.052} C_VEL
LIN {X 0,Y 290.696,Z 251.016,A -85,B 0,C 180,E1 -17252.656,E2 -17252.656} C_VEL
LIN {X 0,Y 289.36,Z 241.512,A -85,B 0,C 180,E1 -17253.982,E2 -17253.982} C_VEL
LIN {X 0,Y 287.332,Z 232.9,A -85,B 0,C 180,E1 -17255.045,E2 -17255.045} C_VEL
LIN {X 0,Y 284.592,Z 223.83,A -85,B 0,C 180,E1 -17256.039,E2 -17256.039} C_VEL
LIN {X 0,Y 283.803,Z 221.104,A -85,B 0,C 180,E1 -17256.326,E2 -17256.326} C_VEL
LIN {X 0,Y 284.192,Z 217.642,A -85,B 0,C 180,E1 -17260.006,E2 -17260.006} C_VEL
LIN {X 0,Y 284.739,Z 213.796,A -85,B 0,C 180,E1 -17264.282,E2 -17264.282} C_VEL
LIN {X 0,Y 284.999,Z 211.363,A -85,B 0,C 180,E1 -17267.179,E2 -17267.179} C_VEL
LIN {X 0,Y 285,Z 208.729,A -85,B 0,C 180,E1 -17270.534,E2 -17270.534} C_VEL
LIN {X 0,Y 284.87,Z 207.021,A -85,B 0,C 180,E1 -17272.916,E2 -17272.916} C_VEL
LIN {X 0,Y 284.622,Z 206.081,A -85,B 0,C 180,E1 -17274.333,E2 -17274.333} C_VEL
LIN {X 0,Y 284.857,Z 205.817,A -85,B 0,C 180,E1 -17278.587,E2 -17278.587} C_VEL
LIN {X 0,Y 284.857,Z 205.813,A -85,B 0,C 180,E1 -17281.415,E2 -17281.415} C_VEL
LIN {X 0,Y 284.676,Z 205.839,A -85,B 0,C 180,E1 -17287.092,E2 -17287.092} C_VEL
LIN {X 0,Y 284.539,Z 205.854,A -85,B 0,C 180,E1 -17289.662,E2 -17289.662} C_VEL
LIN {X 0,Y 283.817,Z 205.947,A -85,B 0,C 180,E1 -17290.842,E2 -17290.842} C_VEL
LIN {X 0,Y 280.987,Z 206.301,A -85,B 0,C 180,E1 -17292.765,E2 -17292.765} C_VEL
LIN {X 0,Y 278.597,Z 206.597,A -85,B 0,C 180,E1 -17294.327,E2 -17294.327} C_VEL
LIN {X 0,Y 277.534,Z 206.728,A -85,B 0,C 180,E1 -17295.536,E2 -17295.536} C_VEL
LIN {X 0,Y 277.425,Z 206.741,A -85,B 0,C 180,E1 -17295.946,E2 -17295.946} C_VEL
LIN {X 0,Y 277.347,Z 206.75,A -85,B 0,C 180,E1 -17300.351,E2 -17300.351} C_VEL
LIN {X 0,Y 277.322,Z 206.755,A -85,B 0,C 180,E1 -17304.171,E2 -17304.171} C_VEL
LIN {X 0,Y 277.328,Z 206.753,A -85,B 0,C 180,E1 -17307.506,E2 -17307.506} C_VEL
LIN {X 0,Y 277.274,Z 206.759,A -85,B 0,C 180,E1 -17310.482,E2 -17310.482} C_VEL
LIN {X 0,Y 277.25,Z 206.761,A -85,B 0,C 180,E1 -17313.896,E2 -17313.896} C_VEL
LIN {X 0,Y 277.274,Z 206.76,A -85,B 0,C 180,E1 -17317.469,E2 -17317.469} C_VEL
LIN {X 0,Y 277.269,Z 206.804,A -85,B 0,C 180,E1 -17320.499,E2 -17320.499} C_VEL
LIN {X 0,Y 277.888,Z 210.372,A -85,B 0,C 180,E1 -17324.916,E2 -17324.916} C_VEL
LIN {X 0,Y 278.639,Z 214.4,A -85,B 0,C 180,E1 -17329.173,E2 -17329.173} C_VEL
LIN {X 0,Y 279.386,Z 218.338,A -85,B 0,C 180,E1 -17332.863,E2 -17332.863} C_VEL
LIN {X 0,Y 280.11,Z 222.63,A -85,B 0,C 180,E1 -17336.497,E2 -17336.497} C_VEL
LIN {X 0,Y 280.036,Z 224.835,A -85,B 0,C 180,E1 -17338.195,E2 -17338.195} C_VEL
LIN {X 0,Y 278.826,Z 230.113,A -85,B 0,C 180,E1 -17341.91,E2 -17341.91} C_VEL
LIN {X 0,Y 277.567,Z 236.342,A -85,B 0,C 180,E1 -17346.102,E2 -17346.102} C_VEL
LIN {X 0,Y 277.363,Z 238.077,A -85,B 0,C 180,E1 -17347.146,E2 -17347.146} C_VEL
LIN {X 0,Y 280.029,Z 249.941,A -85,B 0,C 180,E1 -17348.22,E2 -17348.22} C_VEL
LIN {X 0,Y 281.647,Z 260.582,A -85,B 0,C 180,E1 -17349.394,E2 -17349.394} C_VEL
LIN {X 0,Y 282.211,Z 268.281,A -85,B 0,C 180,E1 -17350.356,E2 -17350.356} C_VEL
LIN {X 0,Y 282.253,Z 276.196,A -85,B 0,C 180,E1 -17351.492,E2 -17351.492} C_VEL
LIN {X 0,Y 281.725,Z 282.85,A -85,B 0,C 180,E1 -17352.581,E2 -17352.581} C_VEL
LIN {X 0,Y 280.297,Z 290.296,A -85,B 0,C 180,E1 -17353.99,E2 -17353.99} C_VEL
LIN {X 0,Y 278.997,Z 296.457,A -85,B 0,C 180,E1 -17355.41,E2 -17355.41} C_VEL
LIN {X 0,Y 278.001,Z 301.587,A -85,B 0,C 180,E1 -17356.849,E2 -17356.849} C_VEL
LIN {X 0,Y 277.146,Z 305.876,A -85,B 0,C 180,E1 -17358.296,E2 -17358.296} C_VEL
LIN {X 0,Y 276.206,Z 311.004,A -85,B 0,C 180,E1 -17360.48,E2 -17360.48} C_VEL
LIN {X 0,Y 275.608,Z 314.751,A -85,B 0,C 180,E1 -17362.675,E2 -17362.675} C_VEL
LIN {X 0,Y 275.364,Z 316.855,A -85,B 0,C 180,E1 -17364.498,E2 -17364.498} C_VEL
LIN {X 0,Y 275.345,Z 318.38,A -85,B 0,C 180,E1 -17367.074,E2 -17367.074} C_VEL
LIN {X 0,Y 275.352,Z 318.615,A -85,B 0,C 180,E1 -17368.538,E2 -17368.538} C_VEL
LIN {X 0,Y 275.412,Z 318.337,A -85,B 0,C 180,E1 -17370,E2 -17370} C_VEL
LIN {X 0,Y 275.383,Z 317.453,A -85,B 0,C 180,E1 -17371.463,E2 -17371.463} C_VEL
LIN {X 0,Y 275.403,Z 316.046,A -85,B 0,C 180,E1 -17372.926,E2 -17372.926} C_VEL
LIN {X 0,Y 275.426,Z 314.102,A -85,B 0,C 180,E1 -17374.391,E2 -17374.391} C_VEL
LIN {X 0,Y 275.42,Z 311.572,A -85,B 0,C 180,E1 -17375.859,E2 -17375.859} C_VEL
LIN {X 0,Y 275.61,Z 308.411,A -85,B 0,C 180,E1 -17377.325,E2 -17377.325} C_VEL
LIN {X 0,Y 275.981,Z 303.351,A -85,B 0,C 180,E1 -17379.158,E2 -17379.158} C_VEL
LIN {X 0,Y 276.399,Z 298.385,A -85,B 0,C 180,E1 -17380.623,E2 -17380.623} C_VEL
LIN {X 0,Y 277.006,Z 292.385,A -85,B 0,C 180,E1 -17382.082,E2 -17382.082} C_VEL
LIN {X 0,Y 277.691,Z 285.06,A -85,B 0,C 180,E1 -17383.539,E2 -17383.539} C_VEL
LIN {X 0,Y 278.459,Z 278.47,A -85,B 0,C 180,E1 -17384.619,E2 -17384.619} C_VEL
LIN {X 0,Y 278.692,Z 273.372,A -85,B 0,C 180,E1 -17385.355,E2 -17385.355} C_VEL
LIN {X 0,Y 278.223,Z 264.023,A -85,B 0,C 180,E1 -17386.472,E2 -17386.472} C_VEL
LIN {X 0,Y 277.575,Z 255.306,A -85,B 0,C 180,E1 -17387.308,E2 -17387.308} C_VEL
LIN {X 0,Y 276.702,Z 245.882,A -85,B 0,C 180,E1 -17388.009,E2 -17388.009} C_VEL
LIN {X 0,Y 276.089,Z 239.474,A -85,B 0,C 180,E1 -17388.41,E2 -17388.41} C_VEL
LIN {X 0,Y 276.939,Z 231.832,A -85,B 0,C 180,E1 -17393.164,E2 -17393.164} C_VEL
LIN {X 0,Y 278.056,Z 224.49,A -85,B 0,C 180,E1 -17397.791,E2 -17397.791} C_VEL
LIN {X 0,Y 279.187,Z 218.069,A -85,B 0,C 180,E1 -17401.914,E2 -17401.914} C_VEL
LIN {X 0,Y 278.702,Z 214.215,A -85,B 0,C 180,E1 -17404.567,E2 -17404.567} C_VEL
LIN {X 0,Y 277.726,Z 208.987,A -85,B 0,C 180,E1 -17408.327,E2 -17408.327} C_VEL
LIN {X 0,Y 277.329,Z 206.758,A -85,B 0,C 180,E1 -17410.046,E2 -17410.046} C_VEL
LIN {X 0,Y 277.205,Z 206.766,A -85,B 0,C 180,E1 -17414.773,E2 -17414.773} C_VEL
LIN {X 0,Y 277.208,Z 206.766,A -85,B 0,C 180,E1 -17418.762,E2 -17418.762} C_VEL
LIN {X 0,Y 277.259,Z 206.76,A -85,B 0,C 180,E1 -17422.528,E2 -17422.528} C_VEL
LIN {X 0,Y 277.25,Z 206.763,A -85,B 0,C 180,E1 -17426.104,E2 -17426.104} C_VEL
LIN {X 0,Y 277.266,Z 206.759,A -85,B 0,C 180,E1 -17429.538,E2 -17429.538} C_VEL
LIN {X 0,Y 277.362,Z 206.744,A -85,B 0,C 180,E1 -17432.863,E2 -17432.863} C_VEL
LIN {X 0,Y 277.302,Z 206.756,A -85,B 0,C 180,E1 -17436.076,E2 -17436.076} C_VEL
LIN {X 0,Y 277.347,Z 206.746,A -85,B 0,C 180,E1 -17440.765,E2 -17440.765} C_VEL
LIN {X 0,Y 277.439,Z 206.739,A -85,B 0,C 180,E1 -17445.325,E2 -17445.325} C_VEL
LIN {X 0,Y 277.461,Z 206.734,A -85,B 0,C 180,E1 -17449.786,E2 -17449.786} C_VEL
LIN {X 0,Y 277.632,Z 206.712,A -85,B 0,C 180,E1 -17452.727,E2 -17452.727} C_VEL
LIN {X 0,Y 277.824,Z 206.687,A -85,B 0,C 180,E1 -17458.549,E2 -17458.549} C_VEL
LIN {X 0,Y 277.823,Z 206.691,A -85,B 0,C 180,E1 -17461.448,E2 -17461.448} C_VEL
LIN {X 0,Y 277.63,Z 206.714,A -85,B 0,C 180,E1 -17467.27,E2 -17467.27} C_VEL
LIN {X 0,Y 277.459,Z 206.734,A -85,B 0,C 180,E1 -17470.212,E2 -17470.212} C_VEL
LIN {X 0,Y 277.41,Z 206.743,A -85,B 0,C 180,E1 -17474.674,E2 -17474.674} C_VEL
LIN {X 0,Y 277.305,Z 206.754,A -85,B 0,C 180,E1 -17479.235,E2 -17479.235} C_VEL
LIN {X 0,Y 277.297,Z 206.753,A -85,B 0,C 180,E1 -17483.922,E2 -17483.922} C_VEL
LIN {X 0,Y 277.325,Z 206.75,A -85,B 0,C 180,E1 -17487.504,E2 -17487.504} C_VEL
LIN {X 0,Y 277.27,Z 206.759,A -85,B 0,C 180,E1 -17490.48,E2 -17490.48} C_VEL
LIN {X 0,Y 277.252,Z 206.761,A -85,B 0,C 180,E1 -17493.893,E2 -17493.893} C_VEL
LIN {X 0,Y 277.278,Z 206.756,A -85,B 0,C 180,E1 -17497.466,E2 -17497.466} C_VEL
LIN {X 0,Y 277.206,Z 206.764,A -85,B 0,C 180,E1 -17501.235,E2 -17501.235} C_VEL
LIN {X 0,Y 277.197,Z 206.766,A -85,B 0,C 180,E1 -17505.225,E2 -17505.225} C_VEL
LIN {X 0,Y 277.218,Z 206.764,A -85,B 0,C 180,E1 -17509.511,E2 -17509.511} C_VEL
LIN {X 0,Y 277.267,Z 206.758,A -85,B 0,C 180,E1 -17512.53,E2 -17512.53} C_VEL
LIN {X 0,Y 277.242,Z 206.761,A -85,B 0,C 180,E1 -17516.103,E2 -17516.103} C_VEL
LIN {X 0,Y 277.255,Z 206.763,A -85,B 0,C 180,E1 -17519.537,E2 -17519.537} C_VEL
LIN {X 0,Y 277.356,Z 206.747,A -85,B 0,C 180,E1 -17522.863,E2 -17522.863} C_VEL
LIN {X 0,Y 277.322,Z 206.75,A -85,B 0,C 180,E1 -17526.079,E2 -17526.079} C_VEL
LIN {X 0,Y 277.338,Z 206.75,A -85,B 0,C 180,E1 -17530.765,E2 -17530.765} C_VEL
LIN {X 0,Y 277.428,Z 206.741,A -85,B 0,C 180,E1 -17535.325,E2 -17535.325} C_VEL
LIN {X 0,Y 277.5,Z 206.728,A -85,B 0,C 180,E1 -17539.788,E2 -17539.788} C_VEL
LIN {X 0,Y 277.645,Z 206.712,A -85,B 0,C 180,E1 -17542.729,E2 -17542.729} C_VEL
LIN {X 0,Y 277.814,Z 206.692,A -85,B 0,C 180,E1 -17548.55,E2 -17548.55} C_VEL
LIN {X 0,Y 277.813,Z 206.689,A -85,B 0,C 180,E1 -17551.449,E2 -17551.449} C_VEL
LIN {X 0,Y 277.653,Z 206.709,A -85,B 0,C 180,E1 -17557.271,E2 -17557.271} C_VEL
LIN {X 0,Y 277.458,Z 206.735,A -85,B 0,C 180,E1 -17560.213,E2 -17560.213} C_VEL
LIN {X 0,Y 277.099,Z 206.78,A -85,B 0,C 180,E1 -17564.692,E2 -17564.692} C_VEL
LIN {X 0,Y 276.885,Z 206.908,A -85,B 0,C 180,E1 -17565.697,E2 -17565.697} C_VEL
LIN {X 0,Y 276.419,Z 211.193,A -85,B 0,C 180,E1 -17569.831,E2 -17569.831} C_VEL
LIN {X 0,Y 276.089,Z 215.661,A -85,B 0,C 180,E1 -17574.034,E2 -17574.034} C_VEL
LIN {X 0,Y 275.843,Z 219.571,A -85,B 0,C 180,E1 -17577.606,E2 -17577.606} C_VEL
LIN {X 0,Y 277.543,Z 229.717,A -85,B 0,C 180,E1 -17578.346,E2 -17578.346} C_VEL
LIN {X 0,Y 278.916,Z 238.885,A -85,B 0,C 180,E1 -17579.222,E2 -17579.222} C_VEL
LIN {X 0,Y 279.735,Z 246.913,A -85,B 0,C 180,E1 -17580.164,E2 -17580.164} C_VEL
LIN {X 0,Y 279.078,Z 254.799,A -85,B 0,C 180,E1 -17581.237,E2 -17581.237} C_VEL
LIN {X 0,Y 278.182,Z 263.406,A -85,B 0,C 180,E1 -17582.685,E2 -17582.685} C_VEL
LIN {X 0,Y 277.347,Z 270.955,A -85,B 0,C 180,E1 -17584.32,E2 -17584.32} C_VEL
LIN {X 0,Y 276.84,Z 276.244,A -85,B 0,C 180,E1 -17585.724,E2 -17585.724} C_VEL
LIN {X 0,Y 276.339,Z 280.732,A -85,B 0,C 180,E1 -17587.158,E2 -17587.158} C_VEL
LIN {X 0,Y 275.901,Z 284.661,A -85,B 0,C 180,E1 -17588.696,E2 -17588.696} C_VEL
LIN {X 0,Y 275.484,Z 288.687,A -85,B 0,C 180,E1 -17590.775,E2 -17590.775} C_VEL
LIN {X 0,Y 275.289,Z 290.786,A -85,B 0,C 180,E1 -17592.241,E2 -17592.241} C_VEL
LIN {X 0,Y 275.158,Z 292.776,A -85,B 0,C 180,E1 -17594.345,E2 -17594.345} C_VEL
LIN {X 0,Y 275.245,Z 293.658,A -85,B 0,C 180,E1 -17596.419,E2 -17596.419} C_VEL
LIN {X 0,Y 275.531,Z 293.489,A -85,B 0,C 180,E1 -17598.459,E2 -17598.459} C_VEL
LIN {X 0,Y 276.033,Z 292.269,A -85,B 0,C 180,E1 -17600.469,E2 -17600.469} C_VEL
LIN {X 0,Y 276.671,Z 290.026,A -85,B 0,C 180,E1 -17602.438,E2 -17602.438} C_VEL
LIN {X 0,Y 277.555,Z 286.733,A -85,B 0,C 180,E1 -17604.384,E2 -17604.384} C_VEL
LIN {X 0,Y 278.305,Z 283.591,A -85,B 0,C 180,E1 -17605.816,E2 -17605.816} C_VEL
LIN {X 0,Y 279.251,Z 279.639,A -85,B 0,C 180,E1 -17607.268,E2 -17607.268} C_VEL
LIN {X 0,Y 280.477,Z 274.064,A -85,B 0,C 180,E1 -17608.907,E2 -17608.907} C_VEL
LIN {X 0,Y 281.808,Z 267.582,A -85,B 0,C 180,E1 -17610.438,E2 -17610.438} C_VEL
LIN {X 0,Y 283.303,Z 259.975,A -85,B 0,C 180,E1 -17611.88,E2 -17611.88} C_VEL
LIN {X 0,Y 284.131,Z 253.338,A -85,B 0,C 180,E1 -17612.931,E2 -17612.931} C_VEL
LIN {X 0,Y 283.004,Z 244.119,A -85,B 0,C 180,E1 -17614.341,E2 -17614.341} C_VEL
LIN {X 0,Y 281.007,Z 235.023,A -85,B 0,C 180,E1 -17615.545,E2 -17615.545} C_VEL
LIN {X 0,Y 278.066,Z 225.319,A -85,B 0,C 180,E1 -17616.682,E2 -17616.682} C_VEL
LIN {X 0,Y 276.83,Z 221.421,A -85,B 0,C 180,E1 -17617.125,E2 -17617.125} C_VEL
LIN {X 0,Y 277.256,Z 218.125,A -85,B 0,C 180,E1 -17620.761,E2 -17620.761} C_VEL
LIN {X 0,Y 277.715,Z 215.228,A -85,B 0,C 180,E1 -17624.08,E2 -17624.08} C_VEL
LIN {X 0,Y 277.978,Z 212.947,A -85,B 0,C 180,E1 -17626.849,E2 -17626.849} C_VEL
LIN {X 0,Y 278.038,Z 210.276,A -85,B 0,C 180,E1 -17630.335,E2 -17630.335} C_VEL
LIN {X 0,Y 277.92,Z 208.582,A -85,B 0,C 180,E1 -17632.737,E2 -17632.737} C_VEL
LIN {X 0,Y 277.468,Z 206.76,A -85,B 0,C 180,E1 -17635.643,E2 -17635.643} C_VEL
LIN {X 0,Y 277.822,Z 206.693,A -85,B 0,C 180,E1 -17638.552,E2 -17638.552} C_VEL
LIN {X 0,Y 277.823,Z 206.689,A -85,B 0,C 180,E1 -17641.451,E2 -17641.451} C_VEL
LIN {X 0,Y 277.63,Z 206.716,A -85,B 0,C 180,E1 -17647.273,E2 -17647.273} C_VEL
LIN {X 0,Y 277.459,Z 206.737,A -85,B 0,C 180,E1 -17650.214,E2 -17650.214} C_VEL
LIN {X 0,Y 277.437,Z 206.739,A -85,B 0,C 180,E1 -17654.675,E2 -17654.675} C_VEL
LIN {X 0,Y 277.425,Z 206.741,A -85,B 0,C 180,E1 -17655.946,E2 -17655.946} C_VEL
LIN {X 0,Y 276.678,Z 206.834,A -85,B 0,C 180,E1 -17657.157,E2 -17657.157} C_VEL
LIN {X 0,Y 273.739,Z 207.199,A -85,B 0,C 180,E1 -17659.13,E2 -17659.13} C_VEL
LIN {X 0,Y 271.3,Z 207.503,A -85,B 0,C 180,E1 -17660.733,E2 -17660.733} C_VEL
LIN {X 0,Y 270.279,Z 207.63,A -85,B 0,C 180,E1 -17661.976,E2 -17661.976} C_VEL
LIN {X 0,Y 270.208,Z 207.637,A -85,B 0,C 180,E1 -17662.398,E2 -17662.398} C_VEL
LIN {X 0,Y 270.266,Z 207.63,A -85,B 0,C 180,E1 -17666.237,E2 -17666.237} C_VEL
LIN {X 0,Y 270.231,Z 207.638,A -85,B 0,C 180,E1 -17669.614,E2 -17669.614} C_VEL
LIN {X 0,Y 270.218,Z 207.638,A -85,B 0,C 180,E1 -17673.667,E2 -17673.667} C_VEL
LIN {X 0,Y 270.23,Z 207.638,A -85,B 0,C 180,E1 -17676.74,E2 -17676.74} C_VEL
LIN {X 0,Y 270.193,Z 207.644,A -85,B 0,C 180,E1 -17679.107,E2 -17679.107} C_VEL
LIN {X 0,Y 270.626,Z 210.074,A -85,B 0,C 180,E1 -17682.471,E2 -17682.471} C_VEL
LIN {X 0,Y 271.22,Z 213.478,A -85,B 0,C 180,E1 -17686.516,E2 -17686.516} C_VEL
LIN {X 0,Y 272.042,Z 217.616,A -85,B 0,C 180,E1 -17690.809,E2 -17690.809} C_VEL
LIN {X 0,Y 272.793,Z 221.706,A -85,B 0,C 180,E1 -17694.574,E2 -17694.574} C_VEL
LIN {X 0,Y 273.241,Z 224.964,A -85,B 0,C 180,E1 -17697.307,E2 -17697.307} C_VEL
LIN {X 0,Y 272.191,Z 229.439,A -85,B 0,C 180,E1 -17700.621,E2 -17700.621} C_VEL
LIN {X 0,Y 270.721,Z 236.158,A -85,B 0,C 180,E1 -17705.316,E2 -17705.316} C_VEL
LIN {X 0,Y 270.47,Z 237.601,A -85,B 0,C 180,E1 -17706.305,E2 -17706.305} C_VEL
LIN {X 0,Y 271.879,Z 243.453,A -85,B 0,C 180,E1 -17706.833,E2 -17706.833} C_VEL
LIN {X 0,Y 273.961,Z 253.449,A -85,B 0,C 180,E1 -17707.875,E2 -17707.875} C_VEL
LIN {X 0,Y 275.259,Z 263.304,A -85,B 0,C 180,E1 -17709.056,E2 -17709.056} C_VEL
LIN {X 0,Y 275.622,Z 274.485,A -85,B 0,C 180,E1 -17710.641,E2 -17710.641} C_VEL
LIN {X 0,Y 275.216,Z 281.854,A -85,B 0,C 180,E1 -17711.868,E2 -17711.868} C_VEL
LIN {X 0,Y 273.896,Z 288.975,A -85,B 0,C 180,E1 -17713.222,E2 -17713.222} C_VEL
LIN {X 0,Y 272.518,Z 295.295,A -85,B 0,C 180,E1 -17714.673,E2 -17714.673} C_VEL
LIN {X 0,Y 271.389,Z 300.567,A -85,B 0,C 180,E1 -17716.141,E2 -17716.141} C_VEL
LIN {X 0,Y 270.186,Z 305.946,A -85,B 0,C 180,E1 -17717.99,E2 -17717.99} C_VEL
LIN {X 0,Y 269.505,Z 309.436,A -85,B 0,C 180,E1 -17719.482,E2 -17719.482} C_VEL
LIN {X 0,Y 268.711,Z 313.487,A -85,B 0,C 180,E1 -17721.73,E2 -17721.73} C_VEL
LIN {X 0,Y 268.307,Z 316.294,A -85,B 0,C 180,E1 -17723.986,E2 -17723.986} C_VEL
LIN {X 0,Y 268.223,Z 317.426,A -85,B 0,C 180,E1 -17725.492,E2 -17725.492} C_VEL
LIN {X 0,Y 268.252,Z 318.078,A -85,B 0,C 180,E1 -17726.997,E2 -17726.997} C_VEL
LIN {X 0,Y 268.275,Z 318.252,A -85,B 0,C 180,E1 -17728.499,E2 -17728.499} C_VEL
LIN {X 0,Y 268.33,Z 317.938,A -85,B 0,C 180,E1 -17730,E2 -17730} C_VEL
LIN {X 0,Y 268.305,Z 317.029,A -85,B 0,C 180,E1 -17731.501,E2 -17731.501} C_VEL
LIN {X 0,Y 268.315,Z 314.683,A -85,B 0,C 180,E1 -17733.755,E2 -17733.755} C_VEL
LIN {X 0,Y 268.35,Z 310.939,A -85,B 0,C 180,E1 -17736.014,E2 -17736.014} C_VEL
LIN {X 0,Y 268.692,Z 305.782,A -85,B 0,C 180,E1 -17738.272,E2 -17738.272} C_VEL
LIN {X 0,Y 269.263,Z 298.899,A -85,B 0,C 180,E1 -17740.528,E2 -17740.528} C_VEL
LIN {X 0,Y 269.863,Z 293.064,A -85,B 0,C 180,E1 -17742.026,E2 -17742.026} C_VEL
LIN {X 0,Y 270.591,Z 285.941,A -85,B 0,C 180,E1 -17743.519,E2 -17743.519} C_VEL
LIN {X 0,Y 271.431,Z 278.36,A -85,B 0,C 180,E1 -17744.815,E2 -17744.815} C_VEL
LIN {X 0,Y 271.634,Z 273.448,A -85,B 0,C 180,E1 -17745.551,E2 -17745.551} C_VEL
LIN {X 0,Y 271.119,Z 263.608,A -85,B 0,C 180,E1 -17746.762,E2 -17746.762} C_VEL
LIN {X 0,Y 270.428,Z 254.137,A -85,B 0,C 180,E1 -17747.683,E2 -17747.683} C_VEL
LIN {X 0,Y 269.471,Z 243.613,A -85,B 0,C 180,E1 -17748.46,E2 -17748.46} C_VEL
LIN {X 0,Y 269.087,Z 239.21,A -85,B 0,C 180,E1 -17748.759,E2 -17748.759} C_VEL
LIN {X 0,Y 269.931,Z 231.493,A -85,B 0,C 180,E1 -17753.701,E2 -17753.701} C_VEL
LIN {X 0,Y 270.976,Z 225.126,A -85,B 0,C 180,E1 -17757.83,E2 -17757.83} C_VEL
LIN {X 0,Y 272.015,Z 219.565,A -85,B 0,C 180,E1 -17761.501,E2 -17761.501} C_VEL
LIN {X 0,Y 272.034,Z 217.595,A -85,B 0,C 180,E1 -17762.857,E2 -17762.857} C_VEL
LIN {X 0,Y 271.174,Z 212.392,A -85,B 0,C 180,E1 -17766.591,E2 -17766.591} C_VEL
LIN {X 0,Y 270.251,Z 207.64,A -85,B 0,C 180,E1 -17770.324,E2 -17770.324} C_VEL
LIN {X 0,Y 270.157,Z 207.645,A -85,B 0,C 180,E1 -17774.62,E2 -17774.62} C_VEL
LIN {X 0,Y 270.169,Z 207.642,A -85,B 0,C 180,E1 -17778.973,E2 -17778.973} C_VEL
LIN {X 0,Y 270.212,Z 207.636,A -85,B 0,C 180,E1 -17781.374,E2 -17781.374} C_VEL
LIN {X 0,Y 270.202,Z 207.636,A -85,B 0,C 180,E1 -17785.093,E2 -17785.093} C_VEL
LIN {X 0,Y 270.205,Z 207.637,A -85,B 0,C 180,E1 -17789.13,E2 -17789.13} C_VEL
LIN {X 0,Y 270.268,Z 207.631,A -85,B 0,C 180,E1 -17792.146,E2 -17792.146} C_VEL
LIN {X 0,Y 270.242,Z 207.634,A -85,B 0,C 180,E1 -17795.537,E2 -17795.537} C_VEL
LIN {X 0,Y 270.305,Z 207.625,A -85,B 0,C 180,E1 -17800.244,E2 -17800.244} C_VEL
LIN {X 0,Y 270.407,Z 207.612,A -85,B 0,C 180,E1 -17804.934,E2 -17804.934} C_VEL
LIN {X 0,Y 270.414,Z 207.614,A -85,B 0,C 180,E1 -17809.517,E2 -17809.517} C_VEL
LIN {X 0,Y 270.588,Z 207.589,A -85,B 0,C 180,E1 -17812.537,E2 -17812.537} C_VEL
LIN {X 0,Y 270.789,Z 207.563,A -85,B 0,C 180,E1 -17818.512,E2 -17818.512} C_VEL
LIN {X 0,Y 270.789,Z 207.567,A -85,B 0,C 180,E1 -17821.486,E2 -17821.486} C_VEL
LIN {X 0,Y 270.587,Z 207.59,A -85,B 0,C 180,E1 -17827.46,E2 -17827.46} C_VEL
LIN {X 0,Y 270.412,Z 207.613,A -85,B 0,C 180,E1 -17830.481,E2 -17830.481} C_VEL
LIN {X 0,Y 270.369,Z 207.618,A -85,B 0,C 180,E1 -17835.065,E2 -17835.065} C_VEL
LIN {X 0,Y 270.252,Z 207.631,A -85,B 0,C 180,E1 -17839.758,E2 -17839.758} C_VEL
LIN {X 0,Y 270.238,Z 207.637,A -85,B 0,C 180,E1 -17844.587,E2 -17844.587} C_VEL
LIN {X 0,Y 270.271,Z 207.63,A -85,B 0,C 180,E1 -17847.907,E2 -17847.907} C_VEL
LIN {X 0,Y 270.183,Z 207.638,A -85,B 0,C 180,E1 -17851.346,E2 -17851.346} C_VEL
LIN {X 0,Y 270.213,Z 207.637,A -85,B 0,C 180,E1 -17854.902,E2 -17854.902} C_VEL
LIN {X 0,Y 270.219,Z 207.635,A -85,B 0,C 180,E1 -17858.715,E2 -17858.715} C_VEL
LIN {X 0,Y 270.161,Z 207.643,A -85,B 0,C 180,E1 -17863.247,E2 -17863.247} C_VEL
LIN {X 0,Y 270.167,Z 207.643,A -85,B 0,C 180,E1 -17867.44,E2 -17867.44} C_VEL
LIN {X 0,Y 270.202,Z 207.639,A -85,B 0,C 180,E1 -17871.373,E2 -17871.373} C_VEL
LIN {X 0,Y 270.197,Z 207.639,A -85,B 0,C 180,E1 -17875.093,E2 -17875.093} C_VEL
LIN {X 0,Y 270.195,Z 207.639,A -85,B 0,C 180,E1 -17879.129,E2 -17879.129} C_VEL
LIN {X 0,Y 270.264,Z 207.63,A -85,B 0,C 180,E1 -17882.142,E2 -17882.142} C_VEL
LIN {X 0,Y 270.271,Z 207.632,A -85,B 0,C 180,E1 -17885.518,E2 -17885.518} C_VEL
LIN {X 0,Y 270.295,Z 207.626,A -85,B 0,C 180,E1 -17890.244,E2 -17890.244} C_VEL
LIN {X 0,Y 270.396,Z 207.615,A -85,B 0,C 180,E1 -17894.935,E2 -17894.935} C_VEL
LIN {X 0,Y 270.435,Z 207.609,A -85,B 0,C 180,E1 -17899.518,E2 -17899.518} C_VEL
LIN {X 0,Y 270.603,Z 207.587,A -85,B 0,C 180,E1 -17902.538,E2 -17902.538} C_VEL
LIN {X 0,Y 270.78,Z 207.568,A -85,B 0,C 180,E1 -17908.512,E2 -17908.512} C_VEL
LIN {X 0,Y 270.779,Z 207.565,A -85,B 0,C 180,E1 -17911.487,E2 -17911.487} C_VEL
LIN {X 0,Y 270.611,Z 207.586,A -85,B 0,C 180,E1 -17917.461,E2 -17917.461} C_VEL
LIN {X 0,Y 270.394,Z 207.618,A -85,B 0,C 180,E1 -17920.483,E2 -17920.483} C_VEL
LIN {X 0,Y 269.99,Z 207.664,A -85,B 0,C 180,E1 -17925.088,E2 -17925.088} C_VEL
LIN {X 0,Y 269.825,Z 207.783,A -85,B 0,C 180,E1 -17925.719,E2 -17925.719} C_VEL
LIN {X 0,Y 269.339,Z 212.259,A -85,B 0,C 180,E1 -17930.06,E2 -17930.06} C_VEL
LIN {X 0,Y 269.053,Z 216.254,A -85,B 0,C 180,E1 -17933.906,E2 -17933.906} C_VEL
LIN {X 0,Y 268.769,Z 219.818,A -85,B 0,C 180,E1 -17937.249,E2 -17937.249} C_VEL
LIN {X 0,Y 270.576,Z 230.542,A -85,B 0,C 180,E1 -17938.085,E2 -17938.085} C_VEL
LIN {X 0,Y 271.909,Z 239.624,A -85,B 0,C 180,E1 -17938.988,E2 -17938.988} C_VEL
LIN {X 0,Y 272.752,Z 247.516,A -85,B 0,C 180,E1 -17939.949,E2 -17939.949} C_VEL
LIN {X 0,Y 272.014,Z 255.778,A -85,B 0,C 180,E1 -17941.113,E2 -17941.113} C_VEL
LIN {X 0,Y 271.1,Z 264.202,A -85,B 0,C 180,E1 -17942.593,E2 -17942.593} C_VEL
LIN {X 0,Y 270.235,Z 271.752,A -85,B 0,C 180,E1 -17944.299,E2 -17944.299} C_VEL
LIN {X 0,Y 269.805,Z 276.222,A -85,B 0,C 180,E1 -17945.51,E2 -17945.51} C_VEL
LIN {X 0,Y 269.318,Z 280.52,A -85,B 0,C 180,E1 -17946.884,E2 -17946.884} C_VEL
LIN {X 0,Y 268.746,Z 285.424,A -85,B 0,C 180,E1 -17948.875,E2 -17948.875} C_VEL
LIN {X 0,Y 268.365,Z 289.168,A -85,B 0,C 180,E1 -17950.897,E2 -17950.897} C_VEL
LIN {X 0,Y 268.119,Z 291.858,A -85,B 0,C 180,E1 -17952.962,E2 -17952.962} C_VEL
LIN {X 0,Y 268.092,Z 293.512,A -85,B 0,C 180,E1 -17955.056,E2 -17955.056} C_VEL
LIN {X 0,Y 268.241,Z 294.082,A -85,B 0,C 180,E1 -17957.19,E2 -17957.19} C_VEL
LIN {X 0,Y 268.648,Z 293.518,A -85,B 0,C 180,E1 -17959.346,E2 -17959.346} C_VEL
LIN {X 0,Y 269.275,Z 291.831,A -85,B 0,C 180,E1 -17961.535,E2 -17961.535} C_VEL
LIN {X 0,Y 269.897,Z 289.744,A -85,B 0,C 180,E1 -17963.21,E2 -17963.21} C_VEL
LIN {X 0,Y 270.896,Z 286.255,A -85,B 0,C 180,E1 -17965.199,E2 -17965.199} C_VEL
LIN {X 0,Y 272.087,Z 281.658,A -85,B 0,C 180,E1 -17967.153,E2 -17967.153} C_VEL
LIN {X 0,Y 273.517,Z 275.683,A -85,B 0,C 180,E1 -17969.078,E2 -17969.078} C_VEL
LIN {X 0,Y 274.832,Z 269.771,A -85,B 0,C 180,E1 -17970.579,E2 -17970.579} C_VEL
LIN {X 0,Y 276.415,Z 262.174,A -85,B 0,C 180,E1 -17972.128,E2 -17972.128} C_VEL
LIN {X 0,Y 277.541,Z 255.111,A -85,B 0,C 180,E1 -17973.316,E2 -17973.316} C_VEL
LIN {X 0,Y 276.705,Z 247.299,A -85,B 0,C 180,E1 -17974.601,E2 -17974.601} C_VEL
LIN {X 0,Y 274.737,Z 237.289,A -85,B 0,C 180,E1 -17976.049,E2 -17976.049} C_VEL
LIN {X 0,Y 271.672,Z 227.248,A -85,B 0,C 180,E1 -17977.32,E2 -17977.32} C_VEL
LIN {X 0,Y 269.912,Z 221.766,A -85,B 0,C 180,E1 -17977.97,E2 -17977.97} C_VEL
LIN {X 0,Y 270.38,Z 218.386,A -85,B 0,C 180,E1 -17981.827,E2 -17981.827} C_VEL
LIN {X 0,Y 270.785,Z 215.781,A -85,B 0,C 180,E1 -17984.959,E2 -17984.959} C_VEL
LIN {X 0,Y 271.041,Z 213.367,A -85,B 0,C 180,E1 -17988.029,E2 -17988.029} C_VEL
LIN {X 0,Y 271.066,Z 211.172,A -85,B 0,C 180,E1 -17991.052,E2 -17991.052} C_VEL
LIN {X 0,Y 270.775,Z 209.234,A -85,B 0,C 180,E1 -17994.042,E2 -17994.042} C_VEL
LIN {X 0,Y 270.631,Z 207.591,A -85,B 0,C 180,E1 -17997.024,E2 -17997.024} C_VEL
LIN {X 0,Y 270.853,Z 207.56,A -85,B 0,C 180,E1 -18000.001,E2 -18000.001} C_VEL
LIN {X 0,Y 270.631,Z 207.584,A -85,B 0,C 180,E1 -18002.978,E2 -18002.978} C_VEL
LIN {X 0,Y 270.587,Z 207.592,A -85,B 0,C 180,E1 -18007.463,E2 -18007.463} C_VEL
LIN {X 0,Y 270.411,Z 207.614,A -85,B 0,C 180,E1 -18010.483,E2 -18010.483} C_VEL
LIN {X 0,Y 270.405,Z 207.616,A -85,B 0,C 180,E1 -18015.066,E2 -18015.066} C_VEL
LIN {X 0,Y 270.304,Z 207.629,A -85,B 0,C 180,E1 -18019.756,E2 -18019.756} C_VEL
LIN {X 0,Y 270.208,Z 207.637,A -85,B 0,C 180,E1 -18022.398,E2 -18022.398} C_VEL
LIN {X 0,Y 269.58,Z 207.719,A -85,B 0,C 180,E1 -18023.642,E2 -18023.642} C_VEL
LIN {X 0,Y 266.772,Z 208.073,A -85,B 0,C 180,E1 -18025.669,E2 -18025.669} C_VEL
LIN {X 0,Y 264.344,Z 208.375,A -85,B 0,C 180,E1 -18027.317,E2 -18027.317} C_VEL
LIN {X 0,Y 263.266,Z 208.504,A -85,B 0,C 180,E1 -18028.594,E2 -18028.594} C_VEL
LIN {X 0,Y 263.16,Z 208.515,A -85,B 0,C 180,E1 -18029.028,E2 -18029.028} C_VEL
LIN {X 0,Y 263.135,Z 208.52,A -85,B 0,C 180,E1 -18032.289,E2 -18032.289} C_VEL
LIN {X 0,Y 263.195,Z 208.514,A -85,B 0,C 180,E1 -18036.767,E2 -18036.767} C_VEL
LIN {X 0,Y 263.165,Z 208.693,A -85,B 0,C 180,E1 -18037.897,E2 -18037.897} C_VEL
LIN {X 0,Y 263.453,Z 209.91,A -85,B 0,C 180,E1 -18039.811,E2 -18039.811} C_VEL
LIN {X 0,Y 263.971,Z 213.033,A -85,B 0,C 180,E1 -18044.04,E2 -18044.04} C_VEL
LIN {X 0,Y 264.643,Z 216.809,A -85,B 0,C 180,E1 -18048.401,E2 -18048.401} C_VEL
LIN {X 0,Y 265.437,Z 220.97,A -85,B 0,C 180,E1 -18052.592,E2 -18052.592} C_VEL
LIN {X 0,Y 266.156,Z 225.104,A -85,B 0,C 180,E1 -18056.323,E2 -18056.323} C_VEL
LIN {X 0,Y 266.022,Z 227.313,A -85,B 0,C 180,E1 -18058.104,E2 -18058.104} C_VEL
LIN {X 0,Y 264.879,Z 231.795,A -85,B 0,C 180,E1 -18061.472,E2 -18061.472} C_VEL
LIN {X 0,Y 263.65,Z 237.285,A -85,B 0,C 180,E1 -18065.401,E2 -18065.401} C_VEL
LIN {X 0,Y 265.129,Z 243.315,A -85,B 0,C 180,E1 -18065.989,E2 -18065.989} C_VEL
LIN {X 0,Y 267.162,Z 252.725,A -85,B 0,C 180,E1 -18067.032,E2 -18067.032} C_VEL
LIN {X 0,Y 268.322,Z 260.736,A -85,B 0,C 180,E1 -18068.017,E2 -18068.017} C_VEL
LIN {X 0,Y 268.91,Z 268.87,A -85,B 0,C 180,E1 -18069.14,E2 -18069.14} C_VEL
LIN {X 0,Y 268.901,Z 276.552,A -85,B 0,C 180,E1 -18070.348,E2 -18070.348} C_VEL
LIN {X 0,Y 268.256,Z 283.934,A -85,B 0,C 180,E1 -18071.676,E2 -18071.676} C_VEL
LIN {X 0,Y 266.331,Z 292.715,A -85,B 0,C 180,E1 -18073.521,E2 -18073.521} C_VEL
LIN {X 0,Y 264.76,Z 299.549,A -85,B 0,C 180,E1 -18075.394,E2 -18075.394} C_VEL
LIN {X 0,Y 263.717,Z 304.084,A -85,B 0,C 180,E1 -18076.908,E2 -18076.908} C_VEL
LIN {X 0,Y 262.841,Z 307.876,A -85,B 0,C 180,E1 -18078.432,E2 -18078.432} C_VEL
LIN {X 0,Y 261.913,Z 312.214,A -85,B 0,C 180,E1 -18080.735,E2 -18080.735} C_VEL
LIN {X 0,Y 261.492,Z 314.442,A -85,B 0,C 180,E1 -18082.277,E2 -18082.277} C_VEL
LIN {X 0,Y 261.173,Z 316.717,A -85,B 0,C 180,E1 -18084.66,E2 -18084.66} C_VEL
LIN {X 0,Y 261.162,Z 317.779,A -85,B 0,C 180,E1 -18086.915,E2 -18086.915} C_VEL
LIN {X 0,Y 261.198,Z 317.887,A -85,B 0,C 180,E1 -18088.458,E2 -18088.458} C_VEL
LIN {X 0,Y 261.25,Z 317.516,A -85,B 0,C 180,E1 -18090,E2 -18090} C_VEL
LIN {X 0,Y 261.229,Z 316.595,A -85,B 0,C 180,E1 -18091.542,E2 -18091.542} C_VEL
LIN {X 0,Y 261.237,Z 314.127,A -85,B 0,C 180,E1 -18093.857,E2 -18093.857} C_VEL
LIN {X 0,Y 261.216,Z 311.735,A -85,B 0,C 180,E1 -18095.44,E2 -18095.44} C_VEL
LIN {X 0,Y 261.506,Z 306.984,A -85,B 0,C 180,E1 -18097.723,E2 -18097.723} C_VEL
LIN {X 0,Y 261.823,Z 302.92,A -85,B 0,C 180,E1 -18099.268,E2 -18099.268} C_VEL
LIN {X 0,Y 262.279,Z 297.998,A -85,B 0,C 180,E1 -18100.811,E2 -18100.811} C_VEL
LIN {X 0,Y 262.87,Z 292.041,A -85,B 0,C 180,E1 -18102.35,E2 -18102.35} C_VEL
LIN {X 0,Y 263.614,Z 284.776,A -85,B 0,C 180,E1 -18103.883,E2 -18103.883} C_VEL
LIN {X 0,Y 264.406,Z 278.251,A -85,B 0,C 180,E1 -18105.02,E2 -18105.02} C_VEL
LIN {X 0,Y 264.543,Z 272.506,A -85,B 0,C 180,E1 -18105.894,E2 -18105.894} C_VEL
LIN {X 0,Y 264.071,Z 263.585,A -85,B 0,C 180,E1 -18107.023,E2 -18107.023} C_VEL
LIN {X 0,Y 263.389,Z 254.194,A -85,B 0,C 180,E1 -18107.97,E2 -18107.97} C_VEL
LIN {X 0,Y 262.502,Z 244.197,A -85,B 0,C 180,E1 -18108.741,E2 -18108.741} C_VEL
LIN {X 0,Y 262.023,Z 238.98,A -85,B 0,C 180,E1 -18109.079,E2 -18109.079} C_VEL
LIN {X 0,Y 262.845,Z 232.073,A -85,B 0,C 180,E1 -18113.646,E2 -18113.646} C_VEL
LIN {X 0,Y 263.869,Z 225.928,A -85,B 0,C 180,E1 -18117.755,E2 -18117.755} C_VEL
LIN {X 0,Y 264.819,Z 220.971,A -85,B 0,C 180,E1 -18121.109,E2 -18121.109} C_VEL
LIN {X 0,Y 264.968,Z 218.342,A -85,B 0,C 180,E1 -18122.939,E2 -18122.939} C_VEL
LIN {X 0,Y 264.364,Z 214.471,A -85,B 0,C 180,E1 -18125.794,E2 -18125.794} C_VEL
LIN {X 0,Y 263.354,Z 209.23,A -85,B 0,C 180,E1 -18129.828,E2 -18129.828} C_VEL
LIN {X 0,Y 263.181,Z 208.52,A -85,B 0,C 180,E1 -18130.611,E2 -18130.611} C_VEL
LIN {X 0,Y 263.127,Z 208.52,A -85,B 0,C 180,E1 -18133.984,E2 -18133.984} C_VEL
LIN {X 0,Y 263.125,Z 208.523,A -85,B 0,C 180,E1 -18138.407,E2 -18138.407} C_VEL
LIN {X 0,Y 263.161,Z 208.518,A -85,B 0,C 180,E1 -18142.102,E2 -18142.102} C_VEL
LIN {X 0,Y 263.156,Z 208.516,A -85,B 0,C 180,E1 -18145.885,E2 -18145.885} C_VEL
LIN {X 0,Y 263.145,Z 208.518,A -85,B 0,C 180,E1 -18149.505,E2 -18149.505} C_VEL
LIN {X 0,Y 263.195,Z 208.509,A -85,B 0,C 180,E1 -18153.002,E2 -18153.002} C_VEL
LIN {X 0,Y 263.159,Z 208.516,A -85,B 0,C 180,E1 -18156.384,E2 -18156.384} C_VEL
LIN {X 0,Y 263.267,Z 208.505,A -85,B 0,C 180,E1 -18159.692,E2 -18159.692} C_VEL
LIN {X 0,Y 263.355,Z 208.49,A -85,B 0,C 180,E1 -18164.521,E2 -18164.521} C_VEL
LIN {X 0,Y 263.357,Z 208.492,A -85,B 0,C 180,E1 -18169.232,E2 -18169.232} C_VEL
LIN {X 0,Y 263.548,Z 208.466,A -85,B 0,C 180,E1 -18172.336,E2 -18172.336} C_VEL
LIN {X 0,Y 263.754,Z 208.439,A -85,B 0,C 180,E1 -18178.472,E2 -18178.472} C_VEL
LIN {X 0,Y 263.753,Z 208.443,A -85,B 0,C 180,E1 -18181.526,E2 -18181.526} C_VEL
LIN {X 0,Y 263.546,Z 208.466,A -85,B 0,C 180,E1 -18187.661,E2 -18187.661} C_VEL
LIN {X 0,Y 263.351,Z 208.495,A -85,B 0,C 180,E1 -18190.765,E2 -18190.765} C_VEL
LIN {X 0,Y 263.311,Z 208.495,A -85,B 0,C 180,E1 -18195.479,E2 -18195.479} C_VEL
LIN {X 0,Y 263.235,Z 208.508,A -85,B 0,C 180,E1 -18200.307,E2 -18200.307} C_VEL
LIN {X 0,Y 263.193,Z 208.51,A -85,B 0,C 180,E1 -18205.291,E2 -18205.291} C_VEL
LIN {X 0,Y 263.179,Z 208.514,A -85,B 0,C 180,E1 -18208.728,E2 -18208.728} C_VEL
LIN {X 0,Y 263.132,Z 208.521,A -85,B 0,C 180,E1 -18212.286,E2 -18212.286} C_VEL
LIN {X 0,Y 263.185,Z 208.514,A -85,B 0,C 180,E1 -18215.976,E2 -18215.976} C_VEL
LIN {X 0,Y 263.112,Z 208.522,A -85,B 0,C 180,E1 -18219.869,E2 -18219.869} C_VEL
LIN {X 0,Y 263.119,Z 208.524,A -85,B 0,C 180,E1 -18223.983,E2 -18223.983} C_VEL
LIN {X 0,Y 263.12,Z 208.519,A -85,B 0,C 180,E1 -18228.405,E2 -18228.405} C_VEL
LIN {X 0,Y 263.179,Z 208.514,A -85,B 0,C 180,E1 -18233.235,E2 -18233.235} C_VEL
LIN {X 0,Y 263.162,Z 208.515,A -85,B 0,C 180,E1 -18235.887,E2 -18235.887} C_VEL
LIN {X 0,Y 263.147,Z 208.52,A -85,B 0,C 180,E1 -18239.506,E2 -18239.506} C_VEL
LIN {X 0,Y 263.191,Z 208.512,A -85,B 0,C 180,E1 -18243.002,E2 -18243.002} C_VEL
LIN {X 0,Y 263.177,Z 208.512,A -85,B 0,C 180,E1 -18246.386,E2 -18246.386} C_VEL
LIN {X 0,Y 263.257,Z 208.504,A -85,B 0,C 180,E1 -18249.692,E2 -18249.692} C_VEL
LIN {X 0,Y 263.344,Z 208.491,A -85,B 0,C 180,E1 -18254.521,E2 -18254.521} C_VEL
LIN {X 0,Y 263.367,Z 208.491,A -85,B 0,C 180,E1 -18259.234,E2 -18259.234} C_VEL
LIN {X 0,Y 263.565,Z 208.463,A -85,B 0,C 180,E1 -18262.338,E2 -18262.338} C_VEL
LIN {X 0,Y 263.744,Z 208.444,A -85,B 0,C 180,E1 -18268.473,E2 -18268.473} C_VEL
LIN {X 0,Y 263.744,Z 208.441,A -85,B 0,C 180,E1 -18271.527,E2 -18271.527} C_VEL
LIN {X 0,Y 263.57,Z 208.463,A -85,B 0,C 180,E1 -18277.661,E2 -18277.661} C_VEL
LIN {X 0,Y 263.316,Z 208.497,A -85,B 0,C 180,E1 -18280.768,E2 -18280.768} C_VEL
LIN {X 0,Y 263.024,Z 208.533,A -85,B 0,C 180,E1 -18283.915,E2 -18283.915} C_VEL
LIN {X 0,Y 262.772,Z 208.6,A -85,B 0,C 180,E1 -18285.675,E2 -18285.675} C_VEL
LIN {X 0,Y 262.223,Z 213.341,A -85,B 0,C 180,E1 -18290.391,E2 -18290.391} C_VEL
LIN {X 0,Y 261.961,Z 217.275,A -85,B 0,C 180,E1 -18294.198,E2 -18294.198} C_VEL
LIN {X 0,Y 261.728,Z 220.139,A -85,B 0,C 180,E1 -18296.945,E2 -18296.945} C_VEL
LIN {X 0,Y 263.604,Z 231.38,A -85,B 0,C 180,E1 -18297.828,E2 -18297.828} C_VEL
LIN {X 0,Y 264.939,Z 240.626,A -85,B 0,C 180,E1 -18298.783,E2 -18298.783} C_VEL
LIN {X 0,Y 265.757,Z 247.744,A -85,B 0,C 180,E1 -18299.682,E2 -18299.682} C_VEL
LIN {X 0,Y 264.984,Z 256.299,A -85,B 0,C 180,E1 -18300.922,E2 -18300.922} C_VEL
LIN {X 0,Y 263.959,Z 265.509,A -85,B 0,C 180,E1 -18302.626,E2 -18302.626} C_VEL
LIN {X 0,Y 263.194,Z 271.946,A -85,B 0,C 180,E1 -18304.131,E2 -18304.131} C_VEL
LIN {X 0,Y 262.669,Z 277.098,A -85,B 0,C 180,E1 -18305.587,E2 -18305.587} C_VEL
LIN {X 0,Y 262.104,Z 281.963,A -85,B 0,C 180,E1 -18307.261,E2 -18307.261} C_VEL
LIN {X 0,Y 261.665,Z 285.693,A -85,B 0,C 180,E1 -18308.842,E2 -18308.842} C_VEL
LIN {X 0,Y 261.383,Z 288.318,A -85,B 0,C 180,E1 -18310.188,E2 -18310.188} C_VEL
LIN {X 0,Y 261.087,Z 291.335,A -85,B 0,C 180,E1 -18312.295,E2 -18312.295} C_VEL
LIN {X 0,Y 261,Z 293.317,A -85,B 0,C 180,E1 -18314.435,E2 -18314.435} C_VEL
LIN {X 0,Y 261.093,Z 294.284,A -85,B 0,C 180,E1 -18316.616,E2 -18316.616} C_VEL
LIN {X 0,Y 261.449,Z 294.199,A -85,B 0,C 180,E1 -18318.822,E2 -18318.822} C_VEL
LIN {X 0,Y 262.041,Z 292.984,A -85,B 0,C 180,E1 -18321.058,E2 -18321.058} C_VEL
LIN {X 0,Y 263.186,Z 289.459,A -85,B 0,C 180,E1 -18324.024,E2 -18324.024} C_VEL
LIN {X 0,Y 264.252,Z 285.812,A -85,B 0,C 180,E1 -18326.049,E2 -18326.049} C_VEL
LIN {X 0,Y 265.606,Z 280.931,A -85,B 0,C 180,E1 -18328.05,E2 -18328.05} C_VEL
LIN {X 0,Y 267.214,Z 274.568,A -85,B 0,C 180,E1 -18330.02,E2 -18330.02} C_VEL
LIN {X 0,Y 268.592,Z 268.565,A -85,B 0,C 180,E1 -18331.512,E2 -18331.512} C_VEL
LIN {X 0,Y 270.132,Z 261.587,A -85,B 0,C 180,E1 -18332.918,E2 -18332.918} C_VEL
LIN {X 0,Y 270.907,Z 256.313,A -85,B 0,C 180,E1 -18333.833,E2 -18333.833} C_VEL
LIN {X 0,Y 270.13,Z 248.369,A -85,B 0,C 180,E1 -18335.197,E2 -18335.197} C_VEL
LIN {X 0,Y 268.315,Z 239.007,A -85,B 0,C 180,E1 -18336.642,E2 -18336.642} C_VEL
LIN {X 0,Y 265.09,Z 228.227,A -85,B 0,C 180,E1 -18338.111,E2 -18338.111} C_VEL
LIN {X 0,Y 263.044,Z 222.359,A -85,B 0,C 180,E1 -18338.839,E2 -18338.839} C_VEL
LIN {X 0,Y 263.03,Z 221.921,A -85,B 0,C 180,E1 -18339.089,E2 -18339.089} C_VEL
LIN {X 0,Y 263.649,Z 218.101,A -85,B 0,C 180,E1 -18343.666,E2 -18343.666} C_VEL
LIN {X 0,Y 264.038,Z 214.974,A -85,B 0,C 180,E1 -18347.707,E2 -18347.707} C_VEL
LIN {X 0,Y 264.109,Z 212.774,A -85,B 0,C 180,E1 -18350.814,E2 -18350.814} C_VEL
LIN {X 0,Y 263.874,Z 210.822,A -85,B 0,C 180,E1 -18353.886,E2 -18353.886} C_VEL
LIN {X 0,Y 263.752,Z 208.446,A -85,B 0,C 180,E1 -18358.474,E2 -18358.474} C_VEL
LIN {X 0,Y 263.752,Z 208.442,A -85,B 0,C 180,E1 -18361.528,E2 -18361.528} C_VEL
LIN {X 0,Y 263.546,Z 208.469,A -85,B 0,C 180,E1 -18367.664,E2 -18367.664} C_VEL
LIN {X 0,Y 263.354,Z 208.494,A -85,B 0,C 180,E1 -18370.768,E2 -18370.768} C_VEL
LIN {X 0,Y 263.353,Z 208.495,A -85,B 0,C 180,E1 -18375.479,E2 -18375.479} C_VEL
LIN {X 0,Y 263.266,Z 208.504,A -85,B 0,C 180,E1 -18380.308,E2 -18380.308} C_VEL
LIN {X 0,Y 263.211,Z 208.506,A -85,B 0,C 180,E1 -18385.292,E2 -18385.292} C_VEL
LIN {X 0,Y 263.16,Z 208.515,A -85,B 0,C 180,E1 -18389.028,E2 -18389.028} C_VEL
LIN {X 0,Y 262.433,Z 208.608,A -85,B 0,C 180,E1 -18390.305,E2 -18390.305} C_VEL
LIN {X 0,Y 259.541,Z 208.968,A -85,B 0,C 180,E1 -18392.387,E2 -18392.387} C_VEL
LIN {X 0,Y 257.152,Z 209.267,A -85,B 0,C 180,E1 -18394.081,E2 -18394.081} C_VEL
LIN {X 0,Y 256.177,Z 209.388,A -85,B 0,C 180,E1 -18395.394,E2 -18395.394} C_VEL
LIN {X 0,Y 256.122,Z 209.395,A -85,B 0,C 180,E1 -18395.839,E2 -18395.839} C_VEL
LIN {X 0,Y 256.586,Z 211.786,A -85,B 0,C 180,E1 -18399.921,E2 -18399.921} C_VEL
LIN {X 0,Y 256.938,Z 214.072,A -85,B 0,C 180,E1 -18403.144,E2 -18403.144} C_VEL
LIN {X 0,Y 257.546,Z 217.593,A -85,B 0,C 180,E1 -18407.459,E2 -18407.459} C_VEL
LIN {X 0,Y 258.25,Z 221.114,A -85,B 0,C 180,E1 -18411.25,E2 -18411.25} C_VEL
LIN {X 0,Y 258.994,Z 225.281,A -85,B 0,C 180,E1 -18415.26,E2 -18415.26} C_VEL
LIN {X 0,Y 259.158,Z 227.51,A -85,B 0,C 180,E1 -18417.213,E2 -18417.213} C_VEL
LIN {X 0,Y 258.443,Z 230.766,A -85,B 0,C 180,E1 -18419.797,E2 -18419.797} C_VEL
LIN {X 0,Y 256.873,Z 236.973,A -85,B 0,C 180,E1 -18424.439,E2 -18424.439} C_VEL
LIN {X 0,Y 257.715,Z 240.258,A -85,B 0,C 180,E1 -18424.758,E2 -18424.758} C_VEL
LIN {X 0,Y 260.247,Z 251.052,A -85,B 0,C 180,E1 -18425.999,E2 -18425.999} C_VEL
LIN {X 0,Y 261.612,Z 259.979,A -85,B 0,C 180,E1 -18427.145,E2 -18427.145} C_VEL
LIN {X 0,Y 262.29,Z 268.531,A -85,B 0,C 180,E1 -18428.381,E2 -18428.381} C_VEL
LIN {X 0,Y 262.315,Z 276.463,A -85,B 0,C 180,E1 -18429.676,E2 -18429.676} C_VEL
LIN {X 0,Y 261.551,Z 284.568,A -85,B 0,C 180,E1 -18431.189,E2 -18431.189} C_VEL
LIN {X 0,Y 259.564,Z 293.084,A -85,B 0,C 180,E1 -18433.078,E2 -18433.078} C_VEL
LIN {X 0,Y 257.889,Z 299.772,A -85,B 0,C 180,E1 -18434.996,E2 -18434.996} C_VEL
LIN {X 0,Y 256.793,Z 304.19,A -85,B 0,C 180,E1 -18436.548,E2 -18436.548} C_VEL
LIN {X 0,Y 255.51,Z 309.426,A -85,B 0,C 180,E1 -18438.899,E2 -18438.899} C_VEL
LIN {X 0,Y 254.631,Z 313.318,A -85,B 0,C 180,E1 -18441.269,E2 -18441.269} C_VEL
LIN {X 0,Y 254.169,Z 315.917,A -85,B 0,C 180,E1 -18443.65,E2 -18443.65} C_VEL
LIN {X 0,Y 254.065,Z 316.969,A -85,B 0,C 180,E1 -18445.24,E2 -18445.24} C_VEL
LIN {X 0,Y 254.075,Z 317.481,A -85,B 0,C 180,E1 -18446.829,E2 -18446.829} C_VEL
LIN {X 0,Y 254.123,Z 317.518,A -85,B 0,C 180,E1 -18448.416,E2 -18448.416} C_VEL
LIN {X 0,Y 254.172,Z 317.075,A -85,B 0,C 180,E1 -18450,E2 -18450} C_VEL
LIN {X 0,Y 254.156,Z 316.12,A -85,B 0,C 180,E1 -18451.585,E2 -18451.585} C_VEL
LIN {X 0,Y 254.159,Z 313.535,A -85,B 0,C 180,E1 -18453.964,E2 -18453.964} C_VEL
LIN {X 0,Y 254.135,Z 311.444,A -85,B 0,C 180,E1 -18455.389,E2 -18455.389} C_VEL
LIN {X 0,Y 254.339,Z 308.102,A -85,B 0,C 180,E1 -18457.143,E2 -18457.143} C_VEL
LIN {X 0,Y 254.711,Z 303.242,A -85,B 0,C 180,E1 -18459.129,E2 -18459.129} C_VEL
LIN {X 0,Y 255.29,Z 297.041,A -85,B 0,C 180,E1 -18461.111,E2 -18461.111} C_VEL
LIN {X 0,Y 255.886,Z 290.957,A -85,B 0,C 180,E1 -18462.693,E2 -18462.693} C_VEL
LIN {X 0,Y 256.577,Z 284.564,A -85,B 0,C 180,E1 -18464.07,E2 -18464.07} C_VEL
LIN {X 0,Y 257.385,Z 278.066,A -85,B 0,C 180,E1 -18465.237,E2 -18465.237} C_VEL
LIN {X 0,Y 257.451,Z 271.506,A -85,B 0,C 180,E1 -18466.251,E2 -18466.251} C_VEL
LIN {X 0,Y 256.997,Z 263.315,A -85,B 0,C 180,E1 -18467.31,E2 -18467.31} C_VEL
LIN {X 0,Y 256.334,Z 253.991,A -85,B 0,C 180,E1 -18468.276,E2 -18468.276} C_VEL
LIN {X 0,Y 255.475,Z 243.99,A -85,B 0,C 180,E1 -18469.068,E2 -18469.068} C_VEL
LIN {X 0,Y 254.963,Z 238.792,A -85,B 0,C 180,E1 -18469.401,E2 -18469.401} C_VEL
LIN {X 0,Y 255.716,Z 232.789,A -85,B 0,C 180,E1 -18473.486,E2 -18473.486} C_VEL
LIN {X 0,Y 256.774,Z 226.602,A -85,B 0,C 180,E1 -18477.73,E2 -18477.73} C_VEL
LIN {X 0,Y 257.76,Z 221.639,A -85,B 0,C 180,E1 -18481.202,E2 -18481.202} C_VEL
LIN {X 0,Y 257.904,Z 219.11,A -85,B 0,C 180,E1 -18483.026,E2 -18483.026} C_VEL
LIN {X 0,Y 257.298,Z 215.207,A -85,B 0,C 180,E1 -18485.963,E2 -18485.963} C_VEL
LIN {X 0,Y 256.148,Z 209.397,A -85,B 0,C 180,E1 -18490.643,E2 -18490.643} C_VEL
LIN {X 0,Y 256.048,Z 209.4,A -85,B 0,C 180,E1 -18495.533,E2 -18495.533} C_VEL
LIN {X 0,Y 256.055,Z 209.401,A -85,B 0,C 180,E1 -18498.795,E2 -18498.795} C_VEL
LIN {X 0,Y 256.13,Z 209.39,A -85,B 0,C 180,E1 -18502.866,E2 -18502.866} C_VEL
LIN {X 0,Y 256.072,Z 209.398,A -85,B 0,C 180,E1 -18506.707,E2 -18506.707} C_VEL
LIN {X 0,Y 256.108,Z 209.394,A -85,B 0,C 180,E1 -18510.398,E2 -18510.398} C_VEL
LIN {X 0,Y 256.175,Z 209.384,A -85,B 0,C 180,E1 -18514.869,E2 -18514.869} C_VEL
LIN {X 0,Y 256.167,Z 209.386,A -85,B 0,C 180,E1 -18519.104,E2 -18519.104} C_VEL
LIN {X 0,Y 256.304,Z 209.37,A -85,B 0,C 180,E1 -18524.084,E2 -18524.084} C_VEL
LIN {X 0,Y 256.3,Z 209.369,A -85,B 0,C 180,E1 -18528.932,E2 -18528.932} C_VEL
LIN {X 0,Y 256.508,Z 209.343,A -85,B 0,C 180,E1 -18532.125,E2 -18532.125} C_VEL
LIN {X 0,Y 256.5,Z 209.345,A -85,B 0,C 180,E1 -18536.857,E2 -18536.857} C_VEL
LIN {X 0,Y 256.76,Z 209.311,A -85,B 0,C 180,E1 -18539.999,E2 -18539.999} C_VEL
LIN {X 0,Y 256.5,Z 209.348,A -85,B 0,C 180,E1 -18543.14,E2 -18543.14} C_VEL
LIN {X 0,Y 256.506,Z 209.343,A -85,B 0,C 180,E1 -18547.873,E2 -18547.873} C_VEL
LIN {X 0,Y 256.292,Z 209.373,A -85,B 0,C 180,E1 -18551.065,E2 -18551.065} C_VEL
LIN {X 0,Y 256.231,Z 209.377,A -85,B 0,C 180,E1 -18555.918,E2 -18555.918} C_VEL
LIN {X 0,Y 256.148,Z 209.39,A -85,B 0,C 180,E1 -18560.895,E2 -18560.895} C_VEL
LIN {X 0,Y 256.17,Z 209.386,A -85,B 0,C 180,E1 -18565.128,E2 -18565.128} C_VEL
LIN {X 0,Y 256.113,Z 209.392,A -85,B 0,C 180,E1 -18569.598,E2 -18569.598} C_VEL
LIN {X 0,Y 256.083,Z 209.395,A -85,B 0,C 180,E1 -18573.288,E2 -18573.288} C_VEL
LIN {X 0,Y 256.125,Z 209.391,A -85,B 0,C 180,E1 -18577.273,E2 -18577.273} C_VEL
LIN {X 0,Y 256.053,Z 209.399,A -85,B 0,C 180,E1 -18581.201,E2 -18581.201} C_VEL
LIN {X 0,Y 256.054,Z 209.402,A -85,B 0,C 180,E1 -18585.529,E2 -18585.529} C_VEL
LIN {X 0,Y 256.05,Z 209.399,A -85,B 0,C 180,E1 -18588.795,E2 -18588.795} C_VEL
LIN {X 0,Y 256.127,Z 209.391,A -85,B 0,C 180,E1 -18592.866,E2 -18592.866} C_VEL
LIN {X 0,Y 256.071,Z 209.396,A -85,B 0,C 180,E1 -18596.707,E2 -18596.707} C_VEL
LIN {X 0,Y 256.137,Z 209.393,A -85,B 0,C 180,E1 -18601.402,E2 -18601.402} C_VEL
LIN {X 0,Y 256.161,Z 209.388,A -85,B 0,C 180,E1 -18605.698,E2 -18605.698} C_VEL
LIN {X 0,Y 256.16,Z 209.39,A -85,B 0,C 180,E1 -18609.104,E2 -18609.104} C_VEL
LIN {X 0,Y 256.293,Z 209.369,A -85,B 0,C 180,E1 -18614.084,E2 -18614.084} C_VEL
LIN {X 0,Y 256.303,Z 209.373,A -85,B 0,C 180,E1 -18618.933,E2 -18618.933} C_VEL
LIN {X 0,Y 256.532,Z 209.338,A -85,B 0,C 180,E1 -18622.127,E2 -18622.127} C_VEL
LIN {X 0,Y 256.707,Z 209.32,A -85,B 0,C 180,E1 -18628.431,E2 -18628.431} C_VEL
LIN {X 0,Y 256.707,Z 209.318,A -85,B 0,C 180,E1 -18631.569,E2 -18631.569} C_VEL
LIN {X 0,Y 256.531,Z 209.34,A -85,B 0,C 180,E1 -18637.873,E2 -18637.873} C_VEL
LIN {X 0,Y 256.243,Z 209.377,A -85,B 0,C 180,E1 -18641.069,E2 -18641.069} C_VEL
LIN {X 0,Y 255.824,Z 209.429,A -85,B 0,C 180,E1 -18645.075,E2 -18645.075} C_VEL
LIN {X 0,Y 255.668,Z 209.724,A -85,B 0,C 180,E1 -18645.955,E2 -18645.955} C_VEL
LIN {X 0,Y 255.089,Z 214.717,A -85,B 0,C 180,E1 -18650.987,E2 -18650.987} C_VEL
LIN {X 0,Y 254.857,Z 218.228,A -85,B 0,C 180,E1 -18654.497,E2 -18654.497} C_VEL
LIN {X 0,Y 254.684,Z 220.364,A -85,B 0,C 180,E1 -18656.587,E2 -18656.587} C_VEL
LIN {X 0,Y 256.584,Z 231.871,A -85,B 0,C 180,E1 -18657.53,E2 -18657.53} C_VEL
LIN {X 0,Y 257.737,Z 239.639,A -85,B 0,C 180,E1 -18658.345,E2 -18658.345} C_VEL
LIN {X 0,Y 258.743,Z 248.486,A -85,B 0,C 180,E1 -18659.483,E2 -18659.483} C_VEL
LIN {X 0,Y 257.811,Z 258.252,A -85,B 0,C 180,E1 -18660.968,E2 -18660.968} C_VEL
LIN {X 0,Y 256.87,Z 266.201,A -85,B 0,C 180,E1 -18662.536,E2 -18662.536} C_VEL
LIN {X 0,Y 256.06,Z 273.01,A -85,B 0,C 180,E1 -18664.201,E2 -18664.201} C_VEL
LIN {X 0,Y 255.351,Z 279.315,A -85,B 0,C 180,E1 -18666.116,E2 -18666.116} C_VEL
LIN {X 0,Y 254.696,Z 285.017,A -85,B 0,C 180,E1 -18668.336,E2 -18668.336} C_VEL
LIN {X 0,Y 254.248,Z 289.084,A -85,B 0,C 180,E1 -18670.511,E2 -18670.511} C_VEL
LIN {X 0,Y 253.954,Z 291.992,A -85,B 0,C 180,E1 -18672.688,E2 -18672.688} C_VEL
LIN {X 0,Y 253.907,Z 293.25,A -85,B 0,C 180,E1 -18673.976,E2 -18673.976} C_VEL
LIN {X 0,Y 253.968,Z 294.47,A -85,B 0,C 180,E1 -18676.228,E2 -18676.228} C_VEL
LIN {X 0,Y 254.281,Z 294.641,A -85,B 0,C 180,E1 -18678.448,E2 -18678.448} C_VEL
LIN {X 0,Y 254.796,Z 293.814,A -85,B 0,C 180,E1 -18680.626,E2 -18680.626} C_VEL
LIN {X 0,Y 255.613,Z 291.904,A -85,B 0,C 180,E1 -18682.877,E2 -18682.877} C_VEL
LIN {X 0,Y 256.727,Z 288.652,A -85,B 0,C 180,E1 -18685.211,E2 -18685.211} C_VEL
LIN {X 0,Y 258.135,Z 283.825,A -85,B 0,C 180,E1 -18687.566,E2 -18687.566} C_VEL
LIN {X 0,Y 259.668,Z 278.532,A -85,B 0,C 180,E1 -18689.516,E2 -18689.516} C_VEL
LIN {X 0,Y 261.615,Z 270.875,A -85,B 0,C 180,E1 -18691.681,E2 -18691.681} C_VEL
LIN {X 0,Y 263.328,Z 263.681,A -85,B 0,C 180,E1 -18693.234,E2 -18693.234} C_VEL
LIN {X 0,Y 264.307,Z 258.535,A -85,B 0,C 180,E1 -18694.191,E2 -18694.191} C_VEL
LIN {X 0,Y 263.815,Z 251.303,A -85,B 0,C 180,E1 -18695.528,E2 -18695.528} C_VEL
LIN {X 0,Y 262.363,Z 242.841,A -85,B 0,C 180,E1 -18696.938,E2 -18696.938} C_VEL
LIN {X 0,Y 260.192,Z 234.511,A -85,B 0,C 180,E1 -18698.2,E2 -18698.2} C_VEL
LIN {X 0,Y 256.628,Z 224.473,A -85,B 0,C 180,E1 -18699.617,E2 -18699.617} C_VEL
LIN {X 0,Y 256.122,Z 222.435,A -85,B 0,C 180,E1 -18699.89,E2 -18699.89} C_VEL
LIN {X 0,Y 256.707,Z 219.031,A -85,B 0,C 180,E1 -18704.113,E2 -18704.113} C_VEL
LIN {X 0,Y 257.019,Z 216.599,A -85,B 0,C 180,E1 -18707.366,E2 -18707.366} C_VEL
LIN {X 0,Y 257.151,Z 214.385,A -85,B 0,C 180,E1 -18710.563,E2 -18710.563} C_VEL
LIN {X 0,Y 256.962,Z 212.426,A -85,B 0,C 180,E1 -18713.721,E2 -18713.721} C_VEL
LIN {X 0,Y 256.778,Z 209.832,A -85,B 0,C 180,E1 -18718.433,E2 -18718.433} C_VEL
LIN {X 0,Y 256.775,Z 209.314,A -85,B 0,C 180,E1 -18720.001,E2 -18720.001} C_VEL
LIN {X 0,Y 256.499,Z 209.344,A -85,B 0,C 180,E1 -18723.143,E2 -18723.143} C_VEL
LIN {X 0,Y 256.506,Z 209.347,A -85,B 0,C 180,E1 -18727.875,E2 -18727.875} C_VEL
LIN {X 0,Y 256.295,Z 209.373,A -85,B 0,C 180,E1 -18732.673,E2 -18732.673} C_VEL
LIN {X 0,Y 256.285,Z 209.374,A -85,B 0,C 180,E1 -18736.303,E2 -18736.303} C_VEL
LIN {X 0,Y 256.16,Z 209.391,A -85,B 0,C 180,E1 -18741.121,E2 -18741.121} C_VEL
LIN {X 0,Y 256.191,Z 209.38,A -85,B 0,C 180,E1 -18745.14,E2 -18745.14} C_VEL
LIN {X 0,Y 256.116,Z 209.396,A -85,B 0,C 180,E1 -18749.601,E2 -18749.601} C_VEL
LIN {X 0,Y 256.07,Z 209.401,A -85,B 0,C 180,E1 -18753.294,E2 -18753.294} C_VEL
LIN {X 0,Y 256.122,Z 209.395,A -85,B 0,C 180,E1 -18755.839,E2 -18755.839} C_VEL
LIN {X 0,Y 255.581,Z 210.238,A -85,B 0,C 180,E1 -18757.149,E2 -18757.149} C_VEL
LIN {X 0,Y 253.033,Z 212.263,A -85,B 0,C 180,E1 -18759.26,E2 -18759.26} C_VEL
LIN {X 0,Y 250.884,Z 214.018,A -85,B 0,C 180,E1 -18760.968,E2 -18760.968} C_VEL
LIN {X 0,Y 250.029,Z 215.14,A -85,B 0,C 180,E1 -18762.294,E2 -18762.294} C_VEL
LIN {X 0,Y 249.999,Z 215.482,A -85,B 0,C 180,E1 -18762.744,E2 -18762.744} C_VEL
LIN {X 0,Y 250.54,Z 218.67,A -85,B 0,C 180,E1 -18766.832,E2 -18766.832} C_VEL
LIN {X 0,Y 251.085,Z 221.375,A -85,B 0,C 180,E1 -18769.926,E2 -18769.926} C_VEL
LIN {X 0,Y 251.848,Z 225.472,A -85,B 0,C 180,E1 -18774.125,E2 -18774.125} C_VEL
LIN {X 0,Y 252.175,Z 228.295,A -85,B 0,C 180,E1 -18776.731,E2 -18776.731} C_VEL
LIN {X 0,Y 251.698,Z 230.877,A -85,B 0,C 180,E1 -18778.898,E2 -18778.898} C_VEL
LIN {X 0,Y 250.124,Z 236.634,A -85,B 0,C 180,E1 -18783.386,E2 -18783.386} C_VEL
LIN {X 0,Y 251.729,Z 242.882,A -85,B 0,C 180,E1 -18784.092,E2 -18784.092} C_VEL
LIN {X 0,Y 254.019,Z 252.932,A -85,B 0,C 180,E1 -18785.353,E2 -18785.353} C_VEL
LIN {X 0,Y 255.434,Z 263.553,A -85,B 0,C 180,E1 -18786.82,E2 -18786.82} C_VEL
LIN {X 0,Y 255.804,Z 273.537,A -85,B 0,C 180,E1 -18788.441,E2 -18788.441} C_VEL
LIN {X 0,Y 255.391,Z 281.231,A -85,B 0,C 180,E1 -18789.877,E2 -18789.877} C_VEL
LIN {X 0,Y 254.486,Z 286.969,A -85,B 0,C 180,E1 -18791.065,E2 -18791.065} C_VEL
LIN {X 0,Y 252.802,Z 293.431,A -85,B 0,C 180,E1 -18792.611,E2 -18792.611} C_VEL
LIN {X 0,Y 251.355,Z 298.831,A -85,B 0,C 180,E1 -18794.18,E2 -18794.18} C_VEL
LIN {X 0,Y 249.883,Z 304.321,A -85,B 0,C 180,E1 -18796.169,E2 -18796.169} C_VEL
LIN {X 0,Y 248.542,Z 309.464,A -85,B 0,C 180,E1 -18798.584,E2 -18798.584} C_VEL
LIN {X 0,Y 247.616,Z 313.248,A -85,B 0,C 180,E1 -18801.019,E2 -18801.019} C_VEL
LIN {X 0,Y 247.087,Z 315.697,A -85,B 0,C 180,E1 -18803.467,E2 -18803.467} C_VEL
LIN {X 0,Y 246.973,Z 316.731,A -85,B 0,C 180,E1 -18805.103,E2 -18805.103} C_VEL
LIN {X 0,Y 246.991,Z 317.184,A -85,B 0,C 180,E1 -18806.738,E2 -18806.738} C_VEL
LIN {X 0,Y 247.049,Z 317.151,A -85,B 0,C 180,E1 -18808.37,E2 -18808.37} C_VEL
LIN {X 0,Y 247.096,Z 316.635,A -85,B 0,C 180,E1 -18810,E2 -18810} C_VEL
LIN {X 0,Y 247.085,Z 315.618,A -85,B 0,C 180,E1 -18811.63,E2 -18811.63} C_VEL
LIN {X 0,Y 247.108,Z 314.031,A -85,B 0,C 180,E1 -18813.261,E2 -18813.261} C_VEL
LIN {X 0,Y 247.112,Z 310.052,A -85,B 0,C 180,E1 -18815.939,E2 -18815.939} C_VEL
LIN {X 0,Y 247.277,Z 307.362,A -85,B 0,C 180,E1 -18817.348,E2 -18817.348} C_VEL
LIN {X 0,Y 247.667,Z 302.366,A -85,B 0,C 180,E1 -18819.391,E2 -18819.391} C_VEL
LIN {X 0,Y 248.127,Z 297.464,A -85,B 0,C 180,E1 -18821.023,E2 -18821.023} C_VEL
LIN {X 0,Y 248.754,Z 291.532,A -85,B 0,C 180,E1 -18822.648,E2 -18822.648} C_VEL
LIN {X 0,Y 249.542,Z 284.297,A -85,B 0,C 180,E1 -18824.267,E2 -18824.267} C_VEL
LIN {X 0,Y 250.368,Z 277.808,A -85,B 0,C 180,E1 -18825.467,E2 -18825.467} C_VEL
LIN {X 0,Y 250.385,Z 271.187,A -85,B 0,C 180,E1 -18826.52,E2 -18826.52} C_VEL
LIN {X 0,Y 249.851,Z 261.754,A -85,B 0,C 180,E1 -18827.756,E2 -18827.756} C_VEL
LIN {X 0,Y 249.202,Z 252.541,A -85,B 0,C 180,E1 -18828.712,E2 -18828.712} C_VEL
LIN {X 0,Y 248.199,Z 241.283,A -85,B 0,C 180,E1 -18829.595,E2 -18829.595} C_VEL
LIN {X 0,Y 247.939,Z 238.506,A -85,B 0,C 180,E1 -18829.778,E2 -18829.778} C_VEL
LIN {X 0,Y 248.762,Z 232.255,A -85,B 0,C 180,E1 -18834.183,E2 -18834.183} C_VEL
LIN {X 0,Y 249.908,Z 226.101,A -85,B 0,C 180,E1 -18838.56,E2 -18838.56} C_VEL
LIN {X 0,Y 250.836,Z 221.109,A -85,B 0,C 180,E1 -18842.165,E2 -18842.165} C_VEL
LIN {X 0,Y 250.383,Z 216.74,A -85,B 0,C 180,E1 -18845.51,E2 -18845.51} C_VEL
LIN {X 0,Y 249.187,Z 210.693,A -85,B 0,C 180,E1 -18850.443,E2 -18850.443} C_VEL
LIN {X 0,Y 249.104,Z 210.271,A -85,B 0,C 180,E1 -18850.993,E2 -18850.993} C_VEL
LIN {X 0,Y 248.997,Z 210.278,A -85,B 0,C 180,E1 -18855.118,E2 -18855.118} C_VEL
LIN {X 0,Y 248.995,Z 210.279,A -85,B 0,C 180,E1 -18859.518,E2 -18859.518} C_VEL
LIN {X 0,Y 249.049,Z 210.273,A -85,B 0,C 180,E1 -18863.657,E2 -18863.657} C_VEL
LIN {X 0,Y 249.042,Z 210.276,A -85,B 0,C 180,E1 -18867.845,E2 -18867.845} C_VEL
LIN {X 0,Y 249.09,Z 210.268,A -85,B 0,C 180,E1 -18871.336,E2 -18871.336} C_VEL
LIN {X 0,Y 249.139,Z 210.261,A -85,B 0,C 180,E1 -18874.966,E2 -18874.966} C_VEL
LIN {X 0,Y 249.113,Z 210.264,A -85,B 0,C 180,E1 -18880.21,E2 -18880.21} C_VEL
LIN {X 0,Y 249.247,Z 210.251,A -85,B 0,C 180,E1 -18883.621,E2 -18883.621} C_VEL
LIN {X 0,Y 249.247,Z 210.247,A -85,B 0,C 180,E1 -18888.615,E2 -18888.615} C_VEL
LIN {X 0,Y 249.45,Z 210.223,A -85,B 0,C 180,E1 -18891.9,E2 -18891.9} C_VEL
LIN {X 0,Y 249.296,Z 210.245,A -85,B 0,C 180,E1 -18895.147,E2 -18895.147} C_VEL
LIN {X 0,Y 249.678,Z 210.192,A -85,B 0,C 180,E1 -18898.386,E2 -18898.386} C_VEL
LIN {X 0,Y 249.678,Z 210.196,A -85,B 0,C 180,E1 -18901.612,E2 -18901.612} C_VEL
LIN {X 0,Y 249.437,Z 210.222,A -85,B 0,C 180,E1 -18906.697,E2 -18906.697} C_VEL
LIN {X 0,Y 249.344,Z 210.236,A -85,B 0,C 180,E1 -18909.735,E2 -18909.735} C_VEL
LIN {X 0,Y 249.173,Z 210.259,A -85,B 0,C 180,E1 -18914.704,E2 -18914.704} C_VEL
LIN {X 0,Y 249.104,Z 210.266,A -85,B 0,C 180,E1 -18918.078,E2 -18918.078} C_VEL
LIN {X 0,Y 249.081,Z 210.268,A -85,B 0,C 180,E1 -18921.517,E2 -18921.517} C_VEL
LIN {X 0,Y 249.117,Z 210.264,A -85,B 0,C 180,E1 -18925.474,E2 -18925.474} C_VEL
LIN {X 0,Y 249.083,Z 210.269,A -85,B 0,C 180,E1 -18928.992,E2 -18928.992} C_VEL
LIN {X 0,Y 249.035,Z 210.277,A -85,B 0,C 180,E1 -18932.423,E2 -18932.423} C_VEL
LIN {X 0,Y 249.067,Z 210.274,A -85,B 0,C 180,E1 -18936.337,E2 -18936.337} C_VEL
LIN {X 0,Y 249.023,Z 210.276,A -85,B 0,C 180,E1 -18940.472,E2 -18940.472} C_VEL
LIN {X 0,Y 248.999,Z 210.279,A -85,B 0,C 180,E1 -18944.878,E2 -18944.878} C_VEL
LIN {X 0,Y 249.012,Z 210.277,A -85,B 0,C 180,E1 -18947.361,E2 -18947.361} C_VEL
LIN {X 0,Y 249.04,Z 210.275,A -85,B 0,C 180,E1 -18952.198,E2 -18952.198} C_VEL
LIN {X 0,Y 249.052,Z 210.275,A -85,B 0,C 180,E1 -18955.64,E2 -18955.64} C_VEL
LIN {X 0,Y 249.048,Z 210.276,A -85,B 0,C 180,E1 -18959.472,E2 -18959.472} C_VEL
LIN {X 0,Y 249.07,Z 210.272,A -85,B 0,C 180,E1 -18963.161,E2 -18963.161} C_VEL
LIN {X 0,Y 249.073,Z 210.269,A -85,B 0,C 180,E1 -18966.732,E2 -18966.732} C_VEL
LIN {X 0,Y 249.104,Z 210.266,A -85,B 0,C 180,E1 -18970.211,E2 -18970.211} C_VEL
LIN {X 0,Y 249.235,Z 210.249,A -85,B 0,C 180,E1 -18973.621,E2 -18973.621} C_VEL
LIN {X 0,Y 249.246,Z 210.25,A -85,B 0,C 180,E1 -18978.616,E2 -18978.616} C_VEL
LIN {X 0,Y 249.474,Z 210.217,A -85,B 0,C 180,E1 -18981.902,E2 -18981.902} C_VEL
LIN {X 0,Y 249.428,Z 210.229,A -85,B 0,C 180,E1 -18986.769,E2 -18986.769} C_VEL
LIN {X 0,Y 249.72,Z 210.187,A -85,B 0,C 180,E1 -18990,E2 -18990} C_VEL
LIN {X 0,Y 249.429,Z 210.226,A -85,B 0,C 180,E1 -18993.23,E2 -18993.23} C_VEL
LIN {X 0,Y 249.456,Z 210.225,A -85,B 0,C 180,E1 -18996.47,E2 -18996.47} C_VEL
LIN {X 0,Y 249.331,Z 210.236,A -85,B 0,C 180,E1 -18999.737,E2 -18999.737} C_VEL
LIN {X 0,Y 248.99,Z 210.281,A -85,B 0,C 180,E1 -19003.05,E2 -19003.05} C_VEL
LIN {X 0,Y 248.635,Z 210.434,A -85,B 0,C 180,E1 -19005.81,E2 -19005.81} C_VEL
LIN {X 0,Y 248.039,Z 215.227,A -85,B 0,C 180,E1 -19010.772,E2 -19010.772} C_VEL
LIN {X 0,Y 247.695,Z 219.61,A -85,B 0,C 180,E1 -19015.189,E2 -19015.189} C_VEL
LIN {X 0,Y 247.625,Z 220.626,A -85,B 0,C 180,E1 -19016.211,E2 -19016.211} C_VEL
LIN {X 0,Y 249.591,Z 232.512,A -85,B 0,C 180,E1 -19017.23,E2 -19017.23} C_VEL
LIN {X 0,Y 250.868,Z 241.393,A -85,B 0,C 180,E1 -19018.213,E2 -19018.213} C_VEL
LIN {X 0,Y 251.727,Z 249.05,A -85,B 0,C 180,E1 -19019.247,E2 -19019.247} C_VEL
LIN {X 0,Y 250.775,Z 258.681,A -85,B 0,C 180,E1 -19020.761,E2 -19020.761} C_VEL
LIN {X 0,Y 249.797,Z 266.865,A -85,B 0,C 180,E1 -19022.434,E2 -19022.434} C_VEL
LIN {X 0,Y 249.1,Z 272.626,A -85,B 0,C 180,E1 -19023.866,E2 -19023.866} C_VEL
LIN {X 0,Y 248.418,Z 278.565,A -85,B 0,C 180,E1 -19025.67,E2 -19025.67} C_VEL
LIN {X 0,Y 247.825,Z 283.283,A -85,B 0,C 180,E1 -19027.438,E2 -19027.438} C_VEL
LIN {X 0,Y 247.255,Z 288.344,A -85,B 0,C 180,E1 -19029.877,E2 -19029.877} C_VEL
LIN {X 0,Y 246.889,Z 291.756,A -85,B 0,C 180,E1 -19032.261,E2 -19032.261} C_VEL
LIN {X 0,Y 246.812,Z 294.393,A -85,B 0,C 180,E1 -19035.388,E2 -19035.388} C_VEL
LIN {X 0,Y 247.044,Z 295.102,A -85,B 0,C 180,E1 -19037.702,E2 -19037.702} C_VEL
LIN {X 0,Y 247.535,Z 294.671,A -85,B 0,C 180,E1 -19040.048,E2 -19040.048} C_VEL
LIN {X 0,Y 248.331,Z 293.091,A -85,B 0,C 180,E1 -19042.413,E2 -19042.413} C_VEL
LIN {X 0,Y 248.83,Z 291.916,A -85,B 0,C 180,E1 -19043.623,E2 -19043.623} C_VEL
LIN {X 0,Y 249.919,Z 288.849,A -85,B 0,C 180,E1 -19045.779,E2 -19045.779} C_VEL
LIN {X 0,Y 251.262,Z 284.661,A -85,B 0,C 180,E1 -19047.899,E2 -19047.899} C_VEL
LIN {X 0,Y 252.92,Z 279.236,A -85,B 0,C 180,E1 -19049.99,E2 -19049.99} C_VEL
LIN {X 0,Y 254.817,Z 272.417,A -85,B 0,C 180,E1 -19052.041,E2 -19052.041} C_VEL
LIN {X 0,Y 256.812,Z 264.612,A -85,B 0,C 180,E1 -19053.816,E2 -19053.816} C_VEL
LIN {X 0,Y 257.798,Z 258.906,A -85,B 0,C 180,E1 -19054.932,E2 -19054.932} C_VEL
LIN {X 0,Y 257.065,Z 250.796,A -85,B 0,C 180,E1 -19056.488,E2 -19056.488} C_VEL
LIN {X 0,Y 255.427,Z 242.126,A -85,B 0,C 180,E1 -19057.984,E2 -19057.984} C_VEL
LIN {X 0,Y 252.774,Z 232.643,A -85,B 0,C 180,E1 -19059.5,E2 -19059.5} C_VEL
LIN {X 0,Y 249.971,Z 225.301,A -85,B 0,C 180,E1 -19060.605,E2 -19060.605} C_VEL
LIN {X 0,Y 249.23,Z 222.776,A -85,B 0,C 180,E1 -19060.972,E2 -19060.972} C_VEL
LIN {X 0,Y 249.673,Z 220.691,A -85,B 0,C 180,E1 -19063.653,E2 -19063.653} C_VEL
LIN {X 0,Y 250.008,Z 218.225,A -85,B 0,C 180,E1 -19067.005,E2 -19067.005} C_VEL
LIN {X 0,Y 250.194,Z 216.005,A -85,B 0,C 180,E1 -19070.298,E2 -19070.298} C_VEL
LIN {X 0,Y 250.04,Z 214.052,A -85,B 0,C 180,E1 -19073.546,E2 -19073.546} C_VEL
LIN {X 0,Y 249.857,Z 211.476,A -85,B 0,C 180,E1 -19078.39,E2 -19078.39} C_VEL
LIN {X 0,Y 249.837,Z 210.71,A -85,B 0,C 180,E1 -19080.001,E2 -19080.001} C_VEL
LIN {X 0,Y 249.677,Z 210.195,A -85,B 0,C 180,E1 -19081.614,E2 -19081.614} C_VEL
LIN {X 0,Y 249.449,Z 210.226,A -85,B 0,C 180,E1 -19086.472,E2 -19086.472} C_VEL
LIN {X 0,Y 249.344,Z 210.24,A -85,B 0,C 180,E1 -19089.738,E2 -19089.738} C_VEL
LIN {X 0,Y 249.207,Z 210.255,A -85,B 0,C 180,E1 -19094.705,E2 -19094.705} C_VEL
LIN {X 0,Y 249.142,Z 210.264,A -85,B 0,C 180,E1 -19098.078,E2 -19098.078} C_VEL
LIN {X 0,Y 249.09,Z 210.27,A -85,B 0,C 180,E1 -19101.519,E2 -19101.519} C_VEL
LIN {X 0,Y 249.133,Z 210.259,A -85,B 0,C 180,E1 -19105.483,E2 -19105.483} C_VEL
LIN {X 0,Y 249.086,Z 210.27,A -85,B 0,C 180,E1 -19108.994,E2 -19108.994} C_VEL
LIN {X 0,Y 249.053,Z 210.273,A -85,B 0,C 180,E1 -19113.903,E2 -19113.903} C_VEL
LIN {X 0,Y 249.457,Z 212.337,A -85,B 0,C 180,E1 -19117.922,E2 -19117.922} C_VEL
LIN {X 0,Y 249.759,Z 213.996,A -85,B 0,C 180,E1 -19120.558,E2 -19120.558} C_VEL
LIN {X 0,Y 249.999,Z 215.482,A -85,B 0,C 180,E1 -19122.744,E2 -19122.744} C_VEL
LIN {X 0,Y 249.502,Z 216.642,A -85,B 0,C 180,E1 -19124.066,E2 -19124.066} C_VEL
LIN {X 0,Y 246.98,Z 219.012,A -85,B 0,C 180,E1 -19126.212,E2 -19126.212} C_VEL
LIN {X 0,Y 244.861,Z 221.006,A -85,B 0,C 180,E1 -19127.953,E2 -19127.953} C_VEL
LIN {X 0,Y 244.071,Z 222.392,A -85,B 0,C 180,E1 -19129.303,E2 -19129.303} C_VEL
LIN {X 0,Y 244.075,Z 222.809,A -85,B 0,C 180,E1 -19129.76,E2 -19129.76} C_VEL
LIN {X 0,Y 244.766,Z 226.31,A -85,B 0,C 180,E1 -19133.512,E2 -19133.512} C_VEL
LIN {X 0,Y 245.211,Z 229.06,A -85,B 0,C 180,E1 -19136.221,E2 -19136.221} C_VEL
LIN {X 0,Y 244.684,Z 232.125,A -85,B 0,C 180,E1 -19138.868,E2 -19138.868} C_VEL
LIN {X 0,Y 243.458,Z 236.299,A -85,B 0,C 180,E1 -19142.258,E2 -19142.258} C_VEL
LIN {X 0,Y 244.313,Z 239.673,A -85,B 0,C 180,E1 -19142.641,E2 -19142.641} C_VEL
LIN {X 0,Y 246.909,Z 250.131,A -85,B 0,C 180,E1 -19144.012,E2 -19144.012} C_VEL
LIN {X 0,Y 248.352,Z 258.765,A -85,B 0,C 180,E1 -19145.248,E2 -19145.248} C_VEL
LIN {X 0,Y 249.138,Z 267.091,A -85,B 0,C 180,E1 -19146.552,E2 -19146.552} C_VEL
LIN {X 0,Y 249.239,Z 274.52,A -85,B 0,C 180,E1 -19147.843,E2 -19147.843} C_VEL
LIN {X 0,Y 248.878,Z 280.857,A -85,B 0,C 180,E1 -19149.075,E2 -19149.075} C_VEL
LIN {X 0,Y 248.205,Z 285.866,A -85,B 0,C 180,E1 -19150.137,E2 -19150.137} C_VEL
LIN {X 0,Y 246.553,Z 292.42,A -85,B 0,C 180,E1 -19151.727,E2 -19151.727} C_VEL
LIN {X 0,Y 244.553,Z 299.086,A -85,B 0,C 180,E1 -19153.728,E2 -19153.728} C_VEL
LIN {X 0,Y 242.989,Z 304.455,A -85,B 0,C 180,E1 -19155.768,E2 -19155.768} C_VEL
LIN {X 0,Y 241.996,Z 307.959,A -85,B 0,C 180,E1 -19157.42,E2 -19157.42} C_VEL
LIN {X 0,Y 240.885,Z 312.027,A -85,B 0,C 180,E1 -19159.918,E2 -19159.918} C_VEL
LIN {X 0,Y 240.347,Z 314.005,A -85,B 0,C 180,E1 -19161.593,E2 -19161.593} C_VEL
LIN {X 0,Y 240.035,Z 315.483,A -85,B 0,C 180,E1 -19163.275,E2 -19163.275} C_VEL
LIN {X 0,Y 239.884,Z 316.474,A -85,B 0,C 180,E1 -19164.958,E2 -19164.958} C_VEL
LIN {X 0,Y 239.889,Z 316.89,A -85,B 0,C 180,E1 -19166.641,E2 -19166.641} C_VEL
LIN {X 0,Y 239.977,Z 316.78,A -85,B 0,C 180,E1 -19168.322,E2 -19168.322} C_VEL
LIN {X 0,Y 240.022,Z 316.189,A -85,B 0,C 180,E1 -19170,E2 -19170} C_VEL
LIN {X 0,Y 240.014,Z 315.098,A -85,B 0,C 180,E1 -19171.678,E2 -19171.678} C_VEL
LIN {X 0,Y 240.022,Z 313.473,A -85,B 0,C 180,E1 -19173.358,E2 -19173.358} C_VEL
LIN {X 0,Y 240.028,Z 309.942,A -85,B 0,C 180,E1 -19175.798,E2 -19175.798} C_VEL
LIN {X 0,Y 240.37,Z 304.681,A -85,B 0,C 180,E1 -19178.407,E2 -19178.407} C_VEL
LIN {X 0,Y 240.833,Z 299.14,A -85,B 0,C 180,E1 -19180.509,E2 -19180.509} C_VEL
LIN {X 0,Y 241.616,Z 292.106,A -85,B 0,C 180,E1 -19182.601,E2 -19182.601} C_VEL
LIN {X 0,Y 242.396,Z 285.044,A -85,B 0,C 180,E1 -19184.268,E2 -19184.268} C_VEL
LIN {X 0,Y 243.355,Z 277.551,A -85,B 0,C 180,E1 -19185.709,E2 -19185.709} C_VEL
LIN {X 0,Y 243.259,Z 269.731,A -85,B 0,C 180,E1 -19186.972,E2 -19186.972} C_VEL
LIN {X 0,Y 242.801,Z 261.715,A -85,B 0,C 180,E1 -19188.046,E2 -19188.046} C_VEL
LIN {X 0,Y 242.139,Z 252.298,A -85,B 0,C 180,E1 -19189.058,E2 -19189.058} C_VEL
LIN {X 0,Y 241.159,Z 241.006,A -85,B 0,C 180,E1 -19189.97,E2 -19189.97} C_VEL
LIN {X 0,Y 240.902,Z 238.263,A -85,B 0,C 180,E1 -19190.159,E2 -19190.159} C_VEL
LIN {X 0,Y 241.865,Z 231.711,A -85,B 0,C 180,E1 -19194.919,E2 -19194.919} C_VEL
LIN {X 0,Y 243.198,Z 224.941,A -85,B 0,C 180,E1 -19199.892,E2 -19199.892} C_VEL
LIN {X 0,Y 243.799,Z 221.825,A -85,B 0,C 180,E1 -19202.229,E2 -19202.229} C_VEL
LIN {X 0,Y 243.38,Z 217.968,A -85,B 0,C 180,E1 -19205.278,E2 -19205.278} C_VEL
LIN {X 0,Y 242.354,Z 212.716,A -85,B 0,C 180,E1 -19209.642,E2 -19209.642} C_VEL
LIN {X 0,Y 242.076,Z 211.146,A -85,B 0,C 180,E1 -19211.102,E2 -19211.102} C_VEL
LIN {X 0,Y 241.926,Z 211.159,A -85,B 0,C 180,E1 -19215.796,E2 -19215.796} C_VEL
LIN {X 0,Y 241.951,Z 211.161,A -85,B 0,C 180,E1 -19220.278,E2 -19220.278} C_VEL
LIN {X 0,Y 241.99,Z 211.151,A -85,B 0,C 180,E1 -19224.488,E2 -19224.488} C_VEL
LIN {X 0,Y 241.978,Z 211.155,A -85,B 0,C 180,E1 -19228.479,E2 -19228.479} C_VEL
LIN {X 0,Y 242.006,Z 211.149,A -85,B 0,C 180,E1 -19232.311,E2 -19232.311} C_VEL
LIN {X 0,Y 242.046,Z 211.148,A -85,B 0,C 180,E1 -19236.013,E2 -19236.013} C_VEL
LIN {X 0,Y 242.04,Z 211.149,A -85,B 0,C 180,E1 -19239.607,E2 -19239.607} C_VEL
LIN {X 0,Y 242.168,Z 211.13,A -85,B 0,C 180,E1 -19243.277,E2 -19243.277} C_VEL
LIN {X 0,Y 242.184,Z 211.127,A -85,B 0,C 180,E1 -19248.278,E2 -19248.278} C_VEL
LIN {X 0,Y 242.397,Z 211.103,A -85,B 0,C 180,E1 -19251.663,E2 -19251.663} C_VEL
LIN {X 0,Y 242.257,Z 211.121,A -85,B 0,C 180,E1 -19255.006,E2 -19255.006} C_VEL
LIN {X 0,Y 242.639,Z 211.069,A -85,B 0,C 180,E1 -19258.339,E2 -19258.339} C_VEL
LIN {X 0,Y 242.638,Z 211.072,A -85,B 0,C 180,E1 -19261.658,E2 -19261.658} C_VEL
LIN {X 0,Y 242.419,Z 211.098,A -85,B 0,C 180,E1 -19266.668,E2 -19266.668} C_VEL
LIN {X 0,Y 242.268,Z 211.117,A -85,B 0,C 180,E1 -19270.022,E2 -19270.022} C_VEL
LIN {X 0,Y 242.128,Z 211.135,A -85,B 0,C 180,E1 -19275.142,E2 -19275.142} C_VEL
LIN {X 0,Y 242.043,Z 211.149,A -85,B 0,C 180,E1 -19278.625,E2 -19278.625} C_VEL
LIN {X 0,Y 242.004,Z 211.151,A -85,B 0,C 180,E1 -19282.179,E2 -19282.179} C_VEL
LIN {X 0,Y 242.066,Z 211.142,A -85,B 0,C 180,E1 -19285.836,E2 -19285.836} C_VEL
LIN {X 0,Y 242.029,Z 211.147,A -85,B 0,C 180,E1 -19289.578,E2 -19289.578} C_VEL
LIN {X 0,Y 241.99,Z 211.151,A -85,B 0,C 180,E1 -19293.489,E2 -19293.489} C_VEL
LIN {X 0,Y 241.999,Z 211.151,A -85,B 0,C 180,E1 -19297.578,E2 -19297.578} C_VEL
LIN {X 0,Y 241.939,Z 211.16,A -85,B 0,C 180,E1 -19301.919,E2 -19301.919} C_VEL
LIN {X 0,Y 241.93,Z 211.159,A -85,B 0,C 180,E1 -19306.57,E2 -19306.57} C_VEL
LIN {X 0,Y 241.952,Z 211.158,A -85,B 0,C 180,E1 -19310.279,E2 -19310.279} C_VEL
LIN {X 0,Y 241.999,Z 211.15,A -85,B 0,C 180,E1 -19314.491,E2 -19314.491} C_VEL
LIN {X 0,Y 241.97,Z 211.154,A -85,B 0,C 180,E1 -19318.479,E2 -19318.479} C_VEL
LIN {X 0,Y 242.006,Z 211.15,A -85,B 0,C 180,E1 -19322.312,E2 -19322.312} C_VEL
LIN {X 0,Y 242.051,Z 211.144,A -85,B 0,C 180,E1 -19326.015,E2 -19326.015} C_VEL
LIN {X 0,Y 242.031,Z 211.149,A -85,B 0,C 180,E1 -19329.607,E2 -19329.607} C_VEL
LIN {X 0,Y 242.157,Z 211.132,A -85,B 0,C 180,E1 -19333.277,E2 -19333.277} C_VEL
LIN {X 0,Y 242.18,Z 211.129,A -85,B 0,C 180,E1 -19338.279,E2 -19338.279} C_VEL
LIN {X 0,Y 242.421,Z 211.096,A -85,B 0,C 180,E1 -19341.665,E2 -19341.665} C_VEL
LIN {X 0,Y 242.252,Z 211.123,A -85,B 0,C 180,E1 -19345.007,E2 -19345.007} C_VEL
LIN {X 0,Y 242.629,Z 211.073,A -85,B 0,C 180,E1 -19348.34,E2 -19348.34} C_VEL
LIN {X 0,Y 242.629,Z 211.071,A -85,B 0,C 180,E1 -19351.66,E2 -19351.66} C_VEL
LIN {X 0,Y 242.427,Z 211.1,A -85,B 0,C 180,E1 -19356.659,E2 -19356.659} C_VEL
LIN {X 0,Y 242.249,Z 211.119,A -85,B 0,C 180,E1 -19360.024,E2 -19360.024} C_VEL
LIN {X 0,Y 241.894,Z 211.164,A -85,B 0,C 180,E1 -19363.44,E2 -19363.44} C_VEL
LIN {X 0,Y 241.56,Z 211.297,A -85,B 0,C 180,E1 -19365.832,E2 -19365.832} C_VEL
LIN {X 0,Y 240.946,Z 216.24,A -85,B 0,C 180,E1 -19371.036,E2 -19371.036} C_VEL
LIN {X 0,Y 240.612,Z 220.881,A -85,B 0,C 180,E1 -19375.858,E2 -19375.858} C_VEL
LIN {X 0,Y 242.253,Z 231.104,A -85,B 0,C 180,E1 -19376.722,E2 -19376.722} C_VEL
LIN {X 0,Y 243.621,Z 240.198,A -85,B 0,C 180,E1 -19377.721,E2 -19377.721} C_VEL
LIN {X 0,Y 244.548,Z 248.031,A -85,B 0,C 180,E1 -19378.775,E2 -19378.775} C_VEL
LIN {X 0,Y 244.437,Z 252.807,A -85,B 0,C 180,E1 -19379.482,E2 -19379.482} C_VEL
LIN {X 0,Y 243.485,Z 261.41,A -85,B 0,C 180,E1 -19381.017,E2 -19381.017} C_VEL
LIN {X 0,Y 242.668,Z 267.762,A -85,B 0,C 180,E1 -19382.397,E2 -19382.397} C_VEL
LIN {X 0,Y 241.935,Z 273.862,A -85,B 0,C 180,E1 -19384,E2 -19384} C_VEL
LIN {X 0,Y 241.315,Z 278.976,A -85,B 0,C 180,E1 -19385.625,E2 -19385.625} C_VEL
LIN {X 0,Y 240.6,Z 284.835,A -85,B 0,C 180,E1 -19387.941,E2 -19387.941} C_VEL
LIN {X 0,Y 240.069,Z 289.467,A -85,B 0,C 180,E1 -19390.437,E2 -19390.437} C_VEL
LIN {X 0,Y 239.746,Z 292.59,A -85,B 0,C 180,E1 -19392.876,E2 -19392.876} C_VEL
LIN {X 0,Y 239.711,Z 294.531,A -85,B 0,C 180,E1 -19395.282,E2 -19395.282} C_VEL
LIN {X 0,Y 239.937,Z 295.38,A -85,B 0,C 180,E1 -19397.65,E2 -19397.65} C_VEL
LIN {X 0,Y 240.42,Z 295.188,A -85,B 0,C 180,E1 -19399.978,E2 -19399.978} C_VEL
LIN {X 0,Y 241.18,Z 293.952,A -85,B 0,C 180,E1 -19402.272,E2 -19402.272} C_VEL
LIN {X 0,Y 242.155,Z 291.706,A -85,B 0,C 180,E1 -19404.52,E2 -19404.52} C_VEL
LIN {X 0,Y 243.456,Z 288.242,A -85,B 0,C 180,E1 -19406.841,E2 -19406.841} C_VEL
LIN {X 0,Y 244.861,Z 284.094,A -85,B 0,C 180,E1 -19408.895,E2 -19408.895} C_VEL
LIN {X 0,Y 246.707,Z 278.459,A -85,B 0,C 180,E1 -19411.036,E2 -19411.036} C_VEL
LIN {X 0,Y 248.802,Z 271.174,A -85,B 0,C 180,E1 -19413.133,E2 -19413.133} C_VEL
LIN {X 0,Y 250.58,Z 264.448,A -85,B 0,C 180,E1 -19414.653,E2 -19414.653} C_VEL
LIN {X 0,Y 251.281,Z 260.742,A -85,B 0,C 180,E1 -19415.417,E2 -19415.417} C_VEL
LIN {X 0,Y 250.608,Z 252.413,A -85,B 0,C 180,E1 -19417.125,E2 -19417.125} C_VEL
LIN {X 0,Y 249.108,Z 243.875,A -85,B 0,C 180,E1 -19418.703,E2 -19418.703} C_VEL
LIN {X 0,Y 247.021,Z 236.08,A -85,B 0,C 180,E1 -19420.039,E2 -19420.039} C_VEL
LIN {X 0,Y 243.655,Z 226.686,A -85,B 0,C 180,E1 -19421.557,E2 -19421.557} C_VEL
LIN {X 0,Y 242.525,Z 223.857,A -85,B 0,C 180,E1 -19422.015,E2 -19422.015} C_VEL
LIN {X 0,Y 242.422,Z 223.11,A -85,B 0,C 180,E1 -19422.171,E2 -19422.171} C_VEL
LIN {X 0,Y 242.803,Z 221.092,A -85,B 0,C 180,E1 -19424.901,E2 -19424.901} C_VEL
LIN {X 0,Y 243.209,Z 218.123,A -85,B 0,C 180,E1 -19429.263,E2 -19429.263} C_VEL
LIN {X 0,Y 243.11,Z 215.679,A -85,B 0,C 180,E1 -19433.361,E2 -19433.361} C_VEL
LIN {X 0,Y 242.947,Z 213.13,A -85,B 0,C 180,E1 -19438.344,E2 -19438.344} C_VEL
LIN {X 0,Y 242.939,Z 212.365,A -85,B 0,C 180,E1 -19440.001,E2 -19440.001} C_VEL
LIN {X 0,Y 242.381,Z 211.163,A -85,B 0,C 180,E1 -19443.326,E2 -19443.326} C_VEL
LIN {X 0,Y 242.419,Z 211.102,A -85,B 0,C 180,E1 -19446.661,E2 -19446.661} C_VEL
LIN {X 0,Y 242.269,Z 211.12,A -85,B 0,C 180,E1 -19450.025,E2 -19450.025} C_VEL
LIN {X 0,Y 242.169,Z 211.133,A -85,B 0,C 180,E1 -19455.142,E2 -19455.142} C_VEL
LIN {X 0,Y 242.076,Z 211.144,A -85,B 0,C 180,E1 -19458.625,E2 -19458.625} C_VEL
LIN {X 0,Y 242.015,Z 211.151,A -85,B 0,C 180,E1 -19462.181,E2 -19462.181} C_VEL
LIN {X 0,Y 242.069,Z 211.139,A -85,B 0,C 180,E1 -19465.839,E2 -19465.839} C_VEL
LIN {X 0,Y 242.033,Z 211.15,A -85,B 0,C 180,E1 -19469.581,E2 -19469.581} C_VEL
LIN {X 0,Y 241.98,Z 211.154,A -85,B 0,C 180,E1 -19471.521,E2 -19471.521} C_VEL
LIN {X 0,Y 242.367,Z 212.981,A -85,B 0,C 180,E1 -19475.716,E2 -19475.716} C_VEL
LIN {X 0,Y 242.739,Z 215.13,A -85,B 0,C 180,E1 -19479.567,E2 -19479.567} C_VEL
LIN {X 0,Y 243.248,Z 218.044,A -85,B 0,C 180,E1 -19483.902,E2 -19483.902} C_VEL
LIN {X 0,Y 243.902,Z 221.723,A -85,B 0,C 180,E1 -19488.521,E2 -19488.521} C_VEL
LIN {X 0,Y 244.075,Z 222.809,A -85,B 0,C 180,E1 -19489.76,E2 -19489.76} C_VEL
LIN {X 0,Y 243.684,Z 224.158,A -85,B 0,C 180,E1 -19491.105,E2 -19491.105} C_VEL
LIN {X 0,Y 241.29,Z 226.809,A -85,B 0,C 180,E1 -19493.288,E2 -19493.288} C_VEL
LIN {X 0,Y 238.438,Z 230.119,A -85,B 0,C 180,E1 -19495.965,E2 -19495.965} C_VEL
LIN {X 0,Y 238.171,Z 231.141,A -85,B 0,C 180,E1 -19496.891,E2 -19496.891} C_VEL
LIN {X 0,Y 237.323,Z 234.461,A -85,B 0,C 180,E1 -19499.773,E2 -19499.773} C_VEL
LIN {X 0,Y 236.814,Z 236.029,A -85,B 0,C 180,E1 -19501.046,E2 -19501.046} C_VEL
LIN {X 0,Y 237.671,Z 239.298,A -85,B 0,C 180,E1 -19501.444,E2 -19501.444} C_VEL
LIN {X 0,Y 240.308,Z 249.554,A -85,B 0,C 180,E1 -19502.888,E2 -19502.888} C_VEL
LIN {X 0,Y 241.88,Z 258.628,A -85,B 0,C 180,E1 -19504.256,E2 -19504.256} C_VEL
LIN {X 0,Y 242.636,Z 267.132,A -85,B 0,C 180,E1 -19505.662,E2 -19505.662} C_VEL
LIN {X 0,Y 242.748,Z 274.366,A -85,B 0,C 180,E1 -19506.993,E2 -19506.993} C_VEL
LIN {X 0,Y 242.265,Z 281.669,A -85,B 0,C 180,E1 -19508.486,E2 -19508.486} C_VEL
LIN {X 0,Y 241.563,Z 286.463,A -85,B 0,C 180,E1 -19509.566,E2 -19509.566} C_VEL
LIN {X 0,Y 239.86,Z 292.86,A -85,B 0,C 180,E1 -19511.198,E2 -19511.198} C_VEL
LIN {X 0,Y 238.128,Z 298.226,A -85,B 0,C 180,E1 -19512.835,E2 -19512.835} C_VEL
LIN {X 0,Y 236.71,Z 302.723,A -85,B 0,C 180,E1 -19514.502,E2 -19514.502} C_VEL
LIN {X 0,Y 235.576,Z 306.487,A -85,B 0,C 180,E1 -19516.192,E2 -19516.192} C_VEL
LIN {X 0,Y 234.214,Z 310.804,A -85,B 0,C 180,E1 -19518.753,E2 -19518.753} C_VEL
LIN {X 0,Y 233.306,Z 313.874,A -85,B 0,C 180,E1 -19521.338,E2 -19521.338} C_VEL
LIN {X 0,Y 232.982,Z 315.269,A -85,B 0,C 180,E1 -19523.07,E2 -19523.07} C_VEL
LIN {X 0,Y 232.782,Z 316.254,A -85,B 0,C 180,E1 -19525.09,E2 -19525.09} C_VEL
LIN {X 0,Y 232.791,Z 316.588,A -85,B 0,C 180,E1 -19526.539,E2 -19526.539} C_VEL
LIN {X 0,Y 232.904,Z 316.407,A -85,B 0,C 180,E1 -19528.271,E2 -19528.271} C_VEL
LIN {X 0,Y 232.95,Z 315.733,A -85,B 0,C 180,E1 -19530,E2 -19530} C_VEL
LIN {X 0,Y 232.945,Z 314.557,A -85,B 0,C 180,E1 -19531.729,E2 -19531.729} C_VEL
LIN {X 0,Y 232.94,Z 312.852,A -85,B 0,C 180,E1 -19533.46,E2 -19533.46} C_VEL
LIN {X 0,Y 232.952,Z 309.213,A -85,B 0,C 180,E1 -19535.975,E2 -19535.975} C_VEL
LIN {X 0,Y 233.167,Z 305.764,A -85,B 0,C 180,E1 -19537.796,E2 -19537.796} C_VEL
LIN {X 0,Y 233.538,Z 301.732,A -85,B 0,C 180,E1 -19539.527,E2 -19539.527} C_VEL
LIN {X 0,Y 233.984,Z 296.831,A -85,B 0,C 180,E1 -19541.259,E2 -19541.259} C_VEL
LIN {X 0,Y 234.655,Z 290.908,A -85,B 0,C 180,E1 -19542.981,E2 -19542.981} C_VEL
LIN {X 0,Y 235.483,Z 283.683,A -85,B 0,C 180,E1 -19544.696,E2 -19544.696} C_VEL
LIN {X 0,Y 236.279,Z 278.433,A -85,B 0,C 180,E1 -19545.749,E2 -19545.749} C_VEL
LIN {X 0,Y 236.236,Z 270.597,A -85,B 0,C 180,E1 -19547.085,E2 -19547.085} C_VEL
LIN {X 0,Y 235.768,Z 262.12,A -85,B 0,C 180,E1 -19548.277,E2 -19548.277} C_VEL
LIN {X 0,Y 235.16,Z 252.974,A -85,B 0,C 180,E1 -19549.306,E2 -19549.306} C_VEL
LIN {X 0,Y 234.292,Z 242.475,A -85,B 0,C 180,E1 -19550.209,E2 -19550.209} C_VEL
LIN {X 0,Y 233.888,Z 237.982,A -85,B 0,C 180,E1 -19550.561,E2 -19550.561} C_VEL
LIN {X 0,Y 235.126,Z 230.401,A -85,B 0,C 180,E1 -19556.269,E2 -19556.269} C_VEL
LIN {X 0,Y 236.533,Z 223.759,A -85,B 0,C 180,E1 -19561.331,E2 -19561.331} C_VEL
LIN {X 0,Y 236.739,Z 222.512,A -85,B 0,C 180,E1 -19562.301,E2 -19562.301} C_VEL
LIN {X 0,Y 236.313,Z 218.677,A -85,B 0,C 180,E1 -19565.423,E2 -19565.423} C_VEL
LIN {X 0,Y 235.261,Z 213.336,A -85,B 0,C 180,E1 -19570.026,E2 -19570.026} C_VEL
LIN {X 0,Y 235.044,Z 212.022,A -85,B 0,C 180,E1 -19571.299,E2 -19571.299} C_VEL
LIN {X 0,Y 234.883,Z 212.038,A -85,B 0,C 180,E1 -19576.512,E2 -19576.512} C_VEL
LIN {X 0,Y 234.922,Z 212.033,A -85,B 0,C 180,E1 -19581.078,E2 -19581.078} C_VEL
LIN {X 0,Y 234.934,Z 212.029,A -85,B 0,C 180,E1 -19585.361,E2 -19585.361} C_VEL
LIN {X 0,Y 234.927,Z 212.033,A -85,B 0,C 180,E1 -19589.43,E2 -19589.43} C_VEL
LIN {X 0,Y 234.998,Z 212.024,A -85,B 0,C 180,E1 -19593.793,E2 -19593.793} C_VEL
LIN {X 0,Y 235.002,Z 212.022,A -85,B 0,C 180,E1 -19598.968,E2 -19598.968} C_VEL
LIN {X 0,Y 235.101,Z 212.009,A -85,B 0,C 180,E1 -19603.058,E2 -19603.058} C_VEL
LIN {X 0,Y 235.118,Z 212.008,A -85,B 0,C 180,E1 -19607.921,E2 -19607.921} C_VEL
LIN {X 0,Y 235.33,Z 211.984,A -85,B 0,C 180,E1 -19611.411,E2 -19611.411} C_VEL
LIN {X 0,Y 235.371,Z 211.979,A -85,B 0,C 180,E1 -19613.139,E2 -19613.139} C_VEL
LIN {X 0,Y 235.598,Z 211.945,A -85,B 0,C 180,E1 -19618.289,E2 -19618.289} C_VEL
LIN {X 0,Y 235.598,Z 211.949,A -85,B 0,C 180,E1 -19621.708,E2 -19621.708} C_VEL
LIN {X 0,Y 235.37,Z 211.977,A -85,B 0,C 180,E1 -19626.858,E2 -19626.858} C_VEL
LIN {X 0,Y 235.214,Z 211.997,A -85,B 0,C 180,E1 -19630.326,E2 -19630.326} C_VEL
LIN {X 0,Y 235.075,Z 212.012,A -85,B 0,C 180,E1 -19635.607,E2 -19635.607} C_VEL
LIN {X 0,Y 234.984,Z 212.026,A -85,B 0,C 180,E1 -19639.206,E2 -19639.206} C_VEL
LIN {X 0,Y 234.951,Z 212.028,A -85,B 0,C 180,E1 -19642.882,E2 -19642.882} C_VEL
LIN {X 0,Y 234.969,Z 212.03,A -85,B 0,C 180,E1 -19646.656,E2 -19646.656} C_VEL
LIN {X 0,Y 234.931,Z 212.032,A -85,B 0,C 180,E1 -19650.566,E2 -19650.566} C_VEL
LIN {X 0,Y 234.959,Z 212.03,A -85,B 0,C 180,E1 -19654.631,E2 -19654.631} C_VEL
LIN {X 0,Y 234.939,Z 212.029,A -85,B 0,C 180,E1 -19658.943,E2 -19658.943} C_VEL
LIN {X 0,Y 234.883,Z 212.038,A -85,B 0,C 180,E1 -19663.484,E2 -19663.484} C_VEL
LIN {X 0,Y 234.883,Z 212.037,A -85,B 0,C 180,E1 -19666.512,E2 -19666.512} C_VEL
LIN {X 0,Y 234.913,Z 212.033,A -85,B 0,C 180,E1 -19671.077,E2 -19671.077} C_VEL
LIN {X 0,Y 234.937,Z 212.032,A -85,B 0,C 180,E1 -19675.363,E2 -19675.363} C_VEL
LIN {X 0,Y 234.927,Z 212.034,A -85,B 0,C 180,E1 -19679.431,E2 -19679.431} C_VEL
LIN {X 0,Y 234.989,Z 212.024,A -85,B 0,C 180,E1 -19683.792,E2 -19683.792} C_VEL
LIN {X 0,Y 235.005,Z 212.024,A -85,B 0,C 180,E1 -19688.969,E2 -19688.969} C_VEL
LIN {X 0,Y 235.09,Z 212.013,A -85,B 0,C 180,E1 -19693.058,E2 -19693.058} C_VEL
LIN {X 0,Y 235.14,Z 212.005,A -85,B 0,C 180,E1 -19697.923,E2 -19697.923} C_VEL
LIN {X 0,Y 235.37,Z 211.975,A -85,B 0,C 180,E1 -19701.413,E2 -19701.413} C_VEL
LIN {X 0,Y 235.397,Z 211.975,A -85,B 0,C 180,E1 -19703.141,E2 -19703.141} C_VEL
LIN {X 0,Y 235.588,Z 211.95,A -85,B 0,C 180,E1 -19708.29,E2 -19708.29} C_VEL
LIN {X 0,Y 235.589,Z 211.948,A -85,B 0,C 180,E1 -19711.709,E2 -19711.709} C_VEL
LIN {X 0,Y 235.396,Z 211.974,A -85,B 0,C 180,E1 -19716.859,E2 -19716.859} C_VEL
LIN {X 0,Y 235.166,Z 212.004,A -85,B 0,C 180,E1 -19720.329,E2 -19720.329} C_VEL
LIN {X 0,Y 234.782,Z 212.051,A -85,B 0,C 180,E1 -19723.855,E2 -19723.855} C_VEL
LIN {X 0,Y 234.483,Z 212.205,A -85,B 0,C 180,E1 -19725.905,E2 -19725.905} C_VEL
LIN {X 0,Y 233.864,Z 217.217,A -85,B 0,C 180,E1 -19731.32,E2 -19731.32} C_VEL
LIN {X 0,Y 233.551,Z 221.17,A -85,B 0,C 180,E1 -19735.482,E2 -19735.482} C_VEL
LIN {X 0,Y 235.317,Z 232.052,A -85,B 0,C 180,E1 -19736.439,E2 -19736.439} C_VEL
LIN {X 0,Y 236.579,Z 240.608,A -85,B 0,C 180,E1 -19737.416,E2 -19737.416} C_VEL
LIN {X 0,Y 237.512,Z 248.384,A -85,B 0,C 180,E1 -19738.499,E2 -19738.499} C_VEL
LIN {X 0,Y 237.427,Z 253.196,A -85,B 0,C 180,E1 -19739.236,E2 -19739.236} C_VEL
LIN {X 0,Y 236.604,Z 260.407,A -85,B 0,C 180,E1 -19740.529,E2 -19740.529} C_VEL
LIN {X 0,Y 235.606,Z 268.118,A -85,B 0,C 180,E1 -19742.234,E2 -19742.234} C_VEL
LIN {X 0,Y 234.871,Z 274.216,A -85,B 0,C 180,E1 -19743.885,E2 -19743.885} C_VEL
LIN {X 0,Y 234.123,Z 280.163,A -85,B 0,C 180,E1 -19745.859,E2 -19745.859} C_VEL
LIN {X 0,Y 233.352,Z 286.248,A -85,B 0,C 180,E1 -19748.462,E2 -19748.462} C_VEL
LIN {X 0,Y 233.031,Z 289.257,A -85,B 0,C 180,E1 -19750.137,E2 -19750.137} C_VEL
LIN {X 0,Y 232.676,Z 292.48,A -85,B 0,C 180,E1 -19752.571,E2 -19752.571} C_VEL
LIN {X 0,Y 232.602,Z 293.911,A -85,B 0,C 180,E1 -19754.022,E2 -19754.022} C_VEL
LIN {X 0,Y 232.71,Z 295.368,A -85,B 0,C 180,E1 -19756.453,E2 -19756.453} C_VEL
LIN {X 0,Y 233.069,Z 295.74,A -85,B 0,C 180,E1 -19758.925,E2 -19758.925} C_VEL
LIN {X 0,Y 233.743,Z 295.041,A -85,B 0,C 180,E1 -19761.42,E2 -19761.42} C_VEL
LIN {X 0,Y 234.768,Z 293.231,A -85,B 0,C 180,E1 -19763.927,E2 -19763.927} C_VEL
LIN {X 0,Y 236.095,Z 290.209,A -85,B 0,C 180,E1 -19766.459,E2 -19766.459} C_VEL
LIN {X 0,Y 237.814,Z 285.654,A -85,B 0,C 180,E1 -19768.983,E2 -19768.983} C_VEL
LIN {X 0,Y 239.352,Z 281.351,A -85,B 0,C 180,E1 -19770.8,E2 -19770.8} C_VEL
LIN {X 0,Y 241.085,Z 275.924,A -85,B 0,C 180,E1 -19772.632,E2 -19772.632} C_VEL
LIN {X 0,Y 242.897,Z 269.876,A -85,B 0,C 180,E1 -19774.28,E2 -19774.28} C_VEL
LIN {X 0,Y 244.734,Z 262.846,A -85,B 0,C 180,E1 -19775.846,E2 -19775.846} C_VEL
LIN {X 0,Y 244.267,Z 254.17,A -85,B 0,C 180,E1 -19777.777,E2 -19777.777} C_VEL
LIN {X 0,Y 242.852,Z 245.685,A -85,B 0,C 180,E1 -19779.448,E2 -19779.448} C_VEL
LIN {X 0,Y 240.531,Z 237.072,A -85,B 0,C 180,E1 -19781.033,E2 -19781.033} C_VEL
LIN {X 0,Y 237.164,Z 227.713,A -85,B 0,C 180,E1 -19782.677,E2 -19782.677} C_VEL
LIN {X 0,Y 235.747,Z 224.204,A -85,B 0,C 180,E1 -19783.282,E2 -19783.282} C_VEL
LIN {X 0,Y 235.613,Z 223.496,A -85,B 0,C 180,E1 -19783.406,E2 -19783.406} C_VEL
LIN {X 0,Y 235.965,Z 221.553,A -85,B 0,C 180,E1 -19786.217,E2 -19786.217} C_VEL
LIN {X 0,Y 236.273,Z 219.27,A -85,B 0,C 180,E1 -19789.721,E2 -19789.721} C_VEL
LIN {X 0,Y 236.173,Z 217.325,A -85,B 0,C 180,E1 -19793.165,E2 -19793.165} C_VEL
LIN {X 0,Y 236.046,Z 214.782,A -85,B 0,C 180,E1 -19798.295,E2 -19798.295} C_VEL
LIN {X 0,Y 236.046,Z 214.044,A -85,B 0,C 180,E1 -19800.001,E2 -19800.001} C_VEL
LIN {X 0,Y 235.484,Z 212.856,A -85,B 0,C 180,E1 -19803.423,E2 -19803.423} C_VEL
LIN {X 0,Y 235.369,Z 211.981,A -85,B 0,C 180,E1 -19806.861,E2 -19806.861} C_VEL
LIN {X 0,Y 235.216,Z 211.998,A -85,B 0,C 180,E1 -19810.329,E2 -19810.329} C_VEL
LIN {X 0,Y 235.116,Z 212.011,A -85,B 0,C 180,E1 -19815.608,E2 -19815.608} C_VEL
LIN {X 0,Y 235.011,Z 212.023,A -85,B 0,C 180,E1 -19819.207,E2 -19819.207} C_VEL
LIN {X 0,Y 234.964,Z 212.03,A -85,B 0,C 180,E1 -19822.884,E2 -19822.884} C_VEL
LIN {X 0,Y 234.972,Z 212.029,A -85,B 0,C 180,E1 -19826.658,E2 -19826.658} C_VEL
LIN {X 0,Y 234.96,Z 212.069,A -85,B 0,C 180,E1 -19828.594,E2 -19828.594} C_VEL
LIN {X 0,Y 235.272,Z 213.707,A -85,B 0,C 180,E1 -19833.237,E2 -19833.237} C_VEL
LIN {X 0,Y 235.568,Z 215.285,A -85,B 0,C 180,E1 -19836.634,E2 -19836.634} C_VEL
